// TIA Portal project "Project2" (V20)

(* hardware
DEVICE "S71500/ET200MP station_1"  S7-1500 station
   slot 0: "Rail_0"  Rack  6ES7 590-1***0-0AA0
   slot 1: "PLC_1"  CPU 1511-1 PN  6ES7 511-1AK00-0AB0  V1.8
      slot 3: "CPU display_1"  6ES7591-1AA00-0AA0
DEVICE "PC-System_1"  SIMATIC PC station
   slot 0: "SIMATIC PC station"  Rail  SIMATIC PC-Station  V1.0
      slot 125: "Stationmanager"  Station_Manager  V6.0.4
   slot 1: "HMI_RT_1"  WinCC RT Advanced  6AV2 104-0xxxx-xxxx  17.0.0.0
      slot 33792: "Computer interface"  Host interface
   slot 2: "IE general_1"  IE General  IE_CP  V8.2.0
      slot 1: "PROFINET interface"  IEGeneral.Interface.8.2.0
*)

// ===== PLC "PLC_1"  CPU 1511-1 PN =====

VAR_GLOBAL   // PLC tag table "Default tag table"
   "Brake_En" AT %M0.0 : Bool;
   "Baffle_Out" AT %MW18 : Int;
   "RPM_In" AT %MW2 : Int;
   "OilTemp_In" AT %MW4 : Int;
   "Baffle_En" AT %M0.1 : Bool;
   "Current_In" AT %MW6 : Int;
   "OilPumpVFDsp_Out" AT %MW8 : Int;
   "OilPumpVFDen_Out" AT %M0.2 : Bool;
   "OilFlow_In" AT %MW10 : Int;
   "TriggerSCL" AT %M0.4 : Bool;
   "Program_Lang" AT %MW12 : Int;
   "Button_LAD" AT %M0.3 : Bool;
   "Button_FBD" AT %M0.5 : Bool;
   "Button_SCL" AT %M0.6 : Bool;
   "Button_STL" AT %M0.7 : Bool;
   "TriggerLAD" AT %M1.0 : Bool;
   "TriggerFBD" AT %M1.1 : Bool;
   "TriggerSTL" AT %M1.2 : Bool;
   "AlarmHorn_En" AT %M1.3 : Bool;
   "StationInterlock_En" AT %M1.4 : Bool;
   "Baffle_Percent" AT %MW14 : Int;
   "OilPumpVFD_percent" AT %MW16 : Int;
   "RPM" AT %MW20 : Int;
   "OilFlow" AT %MW24 : Int;
   "OilTemp" AT %MW28 : Int;
   "Current" AT %MW22 : Int;
   "Static_Test" AT %M1.5 : Bool;
   "BaffleOff_Button" AT %M1.6 : Bool;
   "BaffleHand_Button" AT %M1.7 : Bool;
   "BaffleAuto_Button" AT %M26.0 : Bool;
   "Baffle_HOA" AT %MW70 : Int;
   "SiOff_Button" AT %M26.1 : Bool;
   "StationInterlock_HOA" AT %MW30 : Int;
   "SiHand_Button" AT %M26.2 : Bool;
   "SiAuto_Button" AT %M26.3 : Bool;
   "Brake_HOA" AT %MW40 : Int;
   "BrakeOff_Button" AT %M26.4 : Bool;
   "BrakeHand_Button" AT %M26.5 : Bool;
   "BrakeAuto_Button" AT %M26.6 : Bool;
   "AlarmHorn_HOA" AT %MW50 : Int;
   "AlarmHornOff_Button" AT %M26.7 : Bool;
   "AlarmHornHand_Button" AT %M34.0 : Bool;
   "AlarmHornAuto_Button" AT %M34.1 : Bool;
   "OilPump_HOA" AT %MW60 : Int;
   "OilPumpOff_Button" AT %M34.2 : Bool;
   "OilPumpHand_Button" AT %M34.3 : Bool;
   "OilPumpAuto_Button" AT %M34.4 : Bool;
   "Baffle_Ctrl" AT %M34.5 : Bool;
   "OilPump_Ctrl" AT %M37.0 : Bool;
   "AlarmHorn_Ctrl" AT %M37.1 : Bool;
   "Brake_Ctrl" AT %M37.2 : Bool;
   "StationInterlock_Ctrl" AT %M37.3 : Bool;
   "SeqRunning" AT %M90.0 : Bool;
   "SeqStart" AT %M90.1 : Bool;
   "trigger1" AT %M90.2 : Bool;
   "trigger2" AT %M90.3 : Bool;
   "OverrideVFD_Set" AT %MW92 : Int;
END_VAR

VAR_GLOBAL   // PLC tag table "Alarm_Tags"
   "Overcurrent_set" AT %MW32 : Int;
   "Alarm_Reset" AT %M27.0 : Bool;
   "Alarm_Mute" AT %M27.1 : Bool;
   "OverCurrent_DelaySec" AT %MW38 : Int;
   "OverCurrent_Alarm" AT %M27.2 : Bool;
   "OverCurrent_Horn" AT %M27.3 : Bool;
   "HiOilTemp_DelaySec" AT %MW42 : Int;
   "OilTempMax_set" AT %MW44 : Int;
   "OilTempMax_Horn" AT %M27.4 : Bool;
   "OilTempMax_Alarm" AT %M27.5 : Bool;
   "OverSpeed_DelaySec" AT %MW46 : Int;
   "Overspeed_set" AT %MW48 : Int;
   "OverSpeed_Horn" AT %M27.7 : Bool;
   "OverSpeed_Alarm" AT %M34.6 : Bool;
   "MinOil_set" AT %MW54 : Int;
   "LowOil_Horn" AT %M34.7 : Bool;
   "LowOil_Alarm" AT %M35.0 : Bool;
   "LowOil_DelaySec" AT %MW52 : Int;
   "HighOil_DelaySec" AT %MW56 : Int;
   "MaxOil_set" AT %MW58 : Int;
   "HighOil_Horn" AT %M35.1 : Bool;
   "HighOil_Alarm" AT %M35.2 : Bool;
   "EStop" AT %M35.3 : Bool;
   "EStop_Horn" AT %M35.4 : Bool;
   "EStop_Alarm" AT %M35.5 : Bool;
   "BrakeFail_DelaySec" AT %MW62 : Int;
   "BrakeFail_Horn" AT %M35.6 : Bool;
   "BrakeFail_Alarm" AT %M35.7 : Bool;
END_VAR

VAR_GLOBAL   // PLC tag table "Modes_Tags"
   "WarmupMode" AT %M27.6 : Bool;
   "IdleMode" AT %M36.3 : Bool;
   "GenerationMode" AT %M36.1 : Bool;
   "StabilizeMode" AT %M36.0 : Bool;
   "CooldownMode" AT %M36.2 : Bool;
   "FaultMode" AT %M36.4 : Bool;
   "WarmupRPM" AT %MW64 : Int;
   "Baffel_PID_Set" AT %MW66 : Int;
   "WarmupPumpPct" AT %MW68 : Int;
   "Oilpump_Set" AT %MW72 : Int;
   "WarmupOilTemp" AT %MW74 : Int;
   "WarmupOilTemp_DelaySet" AT %MW76 : Int;
   "WarmupTrans" AT %M36.5 : Bool;
   "Baffel_PID_In" AT %MW78 : Int;
   "Stabile_Current_Set" AT %MW80 : Int;
   "Stabilize_Current_Delay_Set" AT %MW82 : Int;
   "StabilizeTrans" AT %M36.6 : Bool;
   "SystemStop_Button" AT %M36.7 : Bool;
   "GenerationTrans" AT %M37.4 : Bool;
   "SystemStart_Button" AT %M37.5 : Bool;
   "Start_Seq" AT %M37.6 : Bool;
   "CooldownTrans" AT %M37.7 : Bool;
   "CoolDownOilTemp_DelaySet" AT %MW84 : Int;
   "CoolDownRPM_Set" AT %MW86 : Int;
   "CoolDownOilTemp" AT %MW88 : Int;
END_VAR

DATA_BLOCK "SimLogic_DB"   // DB1
{ S7_Optimized_Access := 'TRUE' }
VERSION : 0.1
// stored: InstanceOfName SimLogic
"SimLogic"
BEGIN
END_DATA_BLOCK

DATA_BLOCK "LAD_HOA_DB"   // DB2
{ S7_Optimized_Access := 'TRUE' }
VERSION : 0.1
// stored: InstanceOfName LAD_HOA
"LAD_HOA"
BEGIN
END_DATA_BLOCK

DATA_BLOCK "LAD_IO_DB"   // DB4
{ S7_Optimized_Access := 'TRUE' }
VERSION : 0.1
// stored: InstanceOfName LAD_IO
"LAD_IO"
BEGIN
END_DATA_BLOCK

DATA_BLOCK "FBD_IO_DB"   // DB5
{ S7_Optimized_Access := 'TRUE' }
VERSION : 0.1
// stored: InstanceOfName FBD_IO
"FBD_IO"
BEGIN
END_DATA_BLOCK

DATA_BLOCK "SCL_IO_DB"   // DB6
{ S7_Optimized_Access := 'TRUE' }
VERSION : 0.1
// stored: InstanceOfName SCL_IO
"SCL_IO"
BEGIN
END_DATA_BLOCK

DATA_BLOCK "STL_IO_DB"   // DB7
{ S7_Optimized_Access := 'TRUE' }
VERSION : 0.1
// stored: InstanceOfName STL_IO
"STL_IO"
BEGIN
END_DATA_BLOCK

DATA_BLOCK "FBD_HOA_DB"   // DB8
{ S7_Optimized_Access := 'TRUE' }
VERSION : 0.1
// stored: InstanceOfName FBD_HOA
"FBD_HOA"
BEGIN
END_DATA_BLOCK

DATA_BLOCK "SCL_HOA_DB"   // DB9
{ S7_Optimized_Access := 'TRUE' }
VERSION : 0.1
// stored: InstanceOfName SCL_HOA
"SCL_HOA"
BEGIN
END_DATA_BLOCK

DATA_BLOCK "STL_HOA_DB"   // DB10
{ S7_Optimized_Access := 'TRUE' }
VERSION : 0.1
// stored: InstanceOfName STL_HOA
"STL_HOA"
BEGIN
END_DATA_BLOCK

DATA_BLOCK "LAD_Alarm_DB"   // DB11
{ S7_Optimized_Access := 'TRUE' }
VERSION : 0.1
// stored: InstanceOfName LAD_Alarm
"LAD_Alarm"
BEGIN
END_DATA_BLOCK

DATA_BLOCK "FBD_Alarm_DB"   // DB20
{ S7_Optimized_Access := 'TRUE' }
VERSION : 0.1
// stored: InstanceOfName FBD_Alarm
"FBD_Alarm"
BEGIN
END_DATA_BLOCK

DATA_BLOCK "SCL_Alarm_DB"   // DB21
{ S7_Optimized_Access := 'TRUE' }
VERSION : 0.1
// stored: InstanceOfName SCL_Alarm
"SCL_Alarm"
BEGIN
END_DATA_BLOCK

DATA_BLOCK "STL_Alarm_DB"   // DB22
{ S7_Optimized_Access := 'TRUE' }
VERSION : 0.1
// stored: InstanceOfName STL_Alarm
"STL_Alarm"
BEGIN
END_DATA_BLOCK

DATA_BLOCK "LAD_Modes_DB"   // DB25
{ S7_Optimized_Access := 'TRUE' }
VERSION : 0.1
// stored: InstanceOfName LAD_Modes
"LAD_Modes"
BEGIN
END_DATA_BLOCK

DATA_BLOCK "SEQ_DB"   // DB26
{ S7_Optimized_Access := 'TRUE' }
VERSION : 0.1
// stored: InstanceOfName SEQ
"SEQ"
BEGIN
END_DATA_BLOCK

// folder: System blocks/Program resources

DATA_BLOCK "IEC_Timer_0_DB_25"   // DB3
{ S7_Optimized_Access := 'TRUE' }
AUTHOR : Simatic
FAMILY : IEC
NAME : IEC_TMR
VERSION : 1.0
// stored: InstanceOfName IEC_TIMER
"IEC_TIMER"
BEGIN
END_DATA_BLOCK

DATA_BLOCK "OverCurrent_Tolerance"   // DB12
{ S7_Optimized_Access := 'TRUE' }
AUTHOR : Simatic
FAMILY : IEC
NAME : IEC_TMR
VERSION : 1.0
// stored: InstanceOfName IEC_TIMER
"IEC_TIMER"
BEGIN
END_DATA_BLOCK

DATA_BLOCK "OilTempHi_Tolerance"   // DB13
{ S7_Optimized_Access := 'TRUE' }
AUTHOR : Simatic
FAMILY : IEC
NAME : IEC_TMR
VERSION : 1.0
// stored: InstanceOfName IEC_TIMER
"IEC_TIMER"
BEGIN
END_DATA_BLOCK

DATA_BLOCK "OverSpeed_Tolerance"   // DB14
{ S7_Optimized_Access := 'TRUE' }
AUTHOR : Simatic
FAMILY : IEC
NAME : IEC_TMR
VERSION : 1.0
// stored: InstanceOfName IEC_TIMER
"IEC_TIMER"
BEGIN
END_DATA_BLOCK

DATA_BLOCK "OilLow_Tolerance"   // DB15
{ S7_Optimized_Access := 'TRUE' }
AUTHOR : Simatic
FAMILY : IEC
NAME : IEC_TMR
VERSION : 1.0
// stored: InstanceOfName IEC_TIMER
"IEC_TIMER"
BEGIN
END_DATA_BLOCK

DATA_BLOCK "OilHigh_Tolerance"   // DB16
{ S7_Optimized_Access := 'TRUE' }
AUTHOR : Simatic
FAMILY : IEC
NAME : IEC_TMR
VERSION : 1.0
// stored: InstanceOfName IEC_TIMER
"IEC_TIMER"
BEGIN
END_DATA_BLOCK

DATA_BLOCK "IEC_Timer_0_DB"   // DB17
{ S7_Optimized_Access := 'TRUE' }
AUTHOR : Simatic
FAMILY : IEC
NAME : IEC_TMR
VERSION : 1.0
// stored: InstanceOfName IEC_TIMER
"IEC_TIMER"
BEGIN
END_DATA_BLOCK

DATA_BLOCK "Warmup_to_Stable"   // DB18
{ S7_Optimized_Access := 'TRUE' }
AUTHOR : Simatic
FAMILY : IEC
NAME : IEC_TMR
VERSION : 1.0
// stored: InstanceOfName IEC_TIMER
"IEC_TIMER"
BEGIN
END_DATA_BLOCK

DATA_BLOCK "BrakeFail_Tolerance"   // DB19
{ S7_Optimized_Access := 'TRUE' }
AUTHOR : Simatic
FAMILY : IEC
NAME : IEC_TMR
VERSION : 1.0
// stored: InstanceOfName IEC_TIMER
"IEC_TIMER"
BEGIN
END_DATA_BLOCK

DATA_BLOCK "Stabilize_To_Generation"   // DB23
{ S7_Optimized_Access := 'TRUE' }
AUTHOR : Simatic
FAMILY : IEC
NAME : IEC_TMR
VERSION : 1.0
// stored: InstanceOfName IEC_TIMER
"IEC_TIMER"
BEGIN
END_DATA_BLOCK

DATA_BLOCK "Stable_To_Idle"   // DB24
{ S7_Optimized_Access := 'TRUE' }
AUTHOR : Simatic
FAMILY : IEC
NAME : IEC_TMR
VERSION : 1.0
// stored: InstanceOfName IEC_TIMER
"IEC_TIMER"
BEGIN
END_DATA_BLOCK

DATA_BLOCK "IEC_Timer_1_DB"   // DB43
{ S7_Optimized_Access := 'TRUE' }
AUTHOR : Simatic
FAMILY : IEC
NAME : IEC_TMR
VERSION : 1.0
// stored: InstanceOfName IEC_TIMER
"IEC_TIMER"
BEGIN
END_DATA_BLOCK

// folder: (top level)

FUNCTION_BLOCK "SimLogic"   // FB1, FBD
{ S7_Optimized_Access := 'TRUE' }
VERSION : 0.1
   VAR
      "TO" : Bool;
      rpmv : Int;
      addrpmv : Bool;
      otsp : Int;
      ott : Int;
      TO1 : Bool;
      TO2 : Bool;
      be2 : Int;
      be3 : Int;
      be1 : Int;
      TO3 : Bool;
   END_VAR
   VAR_TEMP
      bf : Int;
      rpmvt : Int;
      bfr : Real;
   END_VAR
BEGIN

REGION Network 1
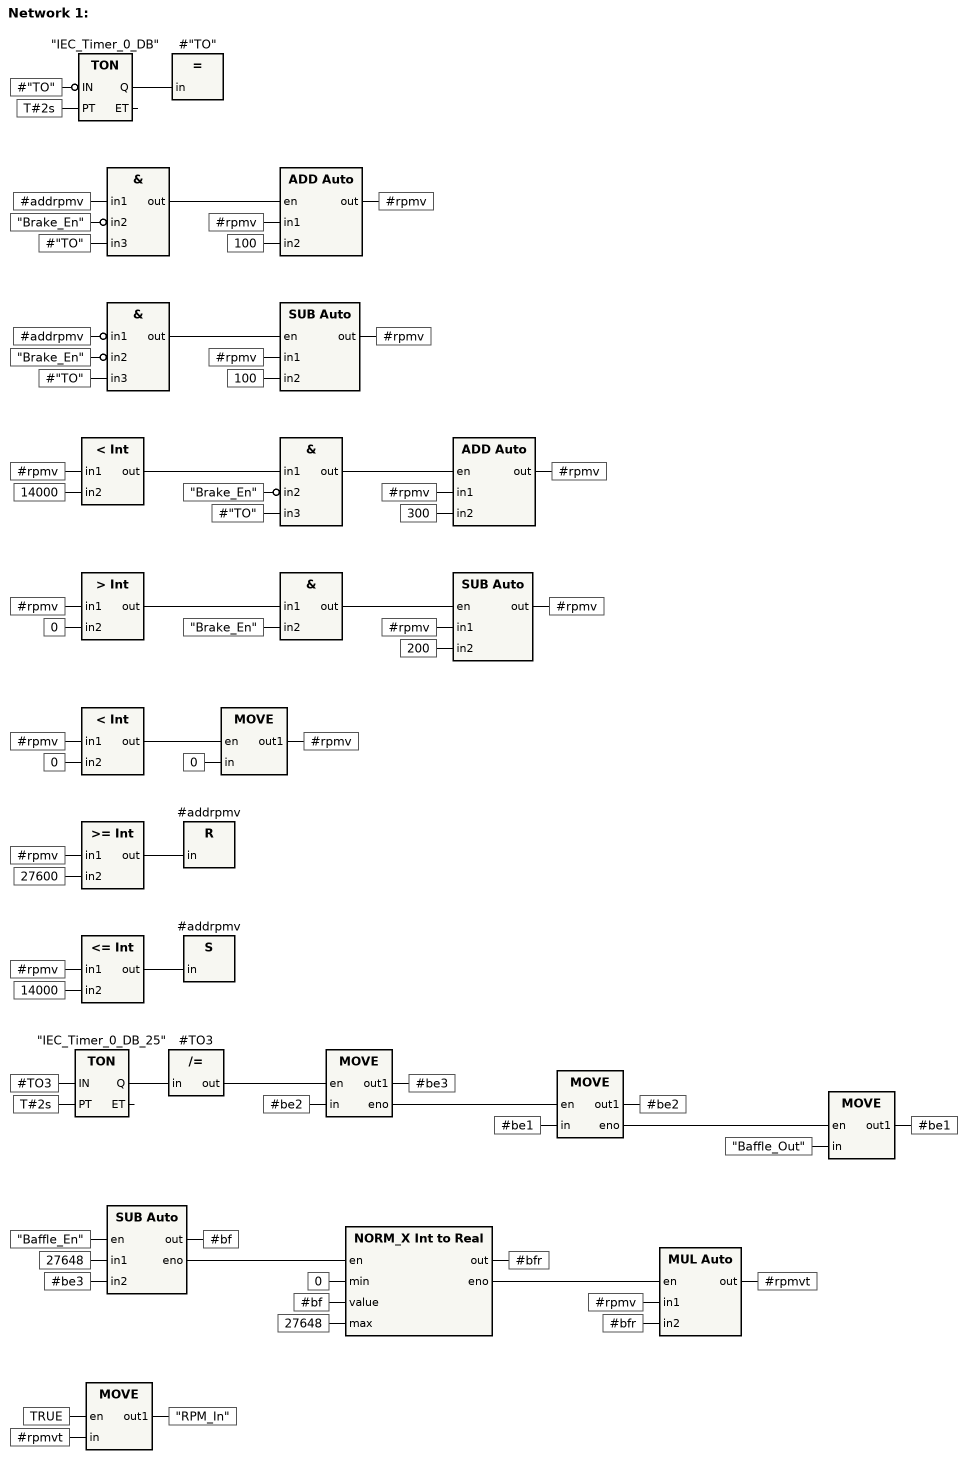
   "IEC_Timer_0_DB".TON(IN := NOT #"TO", PT := T#2s);
   #"TO" := "IEC_Timer_0_DB".Q;
   IF #addrpmv AND NOT "Brake_En" AND #"TO" THEN #rpmv := #rpmv + 100; END_IF;
   IF NOT #addrpmv AND NOT "Brake_En" AND #"TO" THEN #rpmv := #rpmv - 100; END_IF;
   IF (#rpmv < 14000) AND NOT "Brake_En" AND #"TO" THEN #rpmv := #rpmv + 300; END_IF;
   IF (#rpmv > 0) AND "Brake_En" THEN #rpmv := #rpmv - 200; END_IF;
   IF #rpmv < 0 THEN #rpmv := 0; END_IF;
   IF #rpmv >= 27600 THEN #addrpmv := FALSE; END_IF;
   IF #rpmv <= 14000 THEN #addrpmv := TRUE; END_IF;
   "IEC_Timer_0_DB_25".TON(IN := #TO3, PT := T#2s);
   #TO3 := NOT "IEC_Timer_0_DB_25".Q;
   IF "IEC_Timer_0_DB_25".Q THEN
       #be3 := #be2;
       #be2 := #be1;
       #be1 := "Baffle_Out";
   END_IF;
   IF "Baffle_En" THEN
       #bf := 27648 - #be3;
       #bfr := NORM_X(MIN := 0, VALUE := #bf, MAX := 27648);
       #rpmvt := #rpmv * #bfr;
   END_IF;
   IF TRUE THEN "RPM_In" := #rpmvt; END_IF;
END_REGION

REGION Network 2
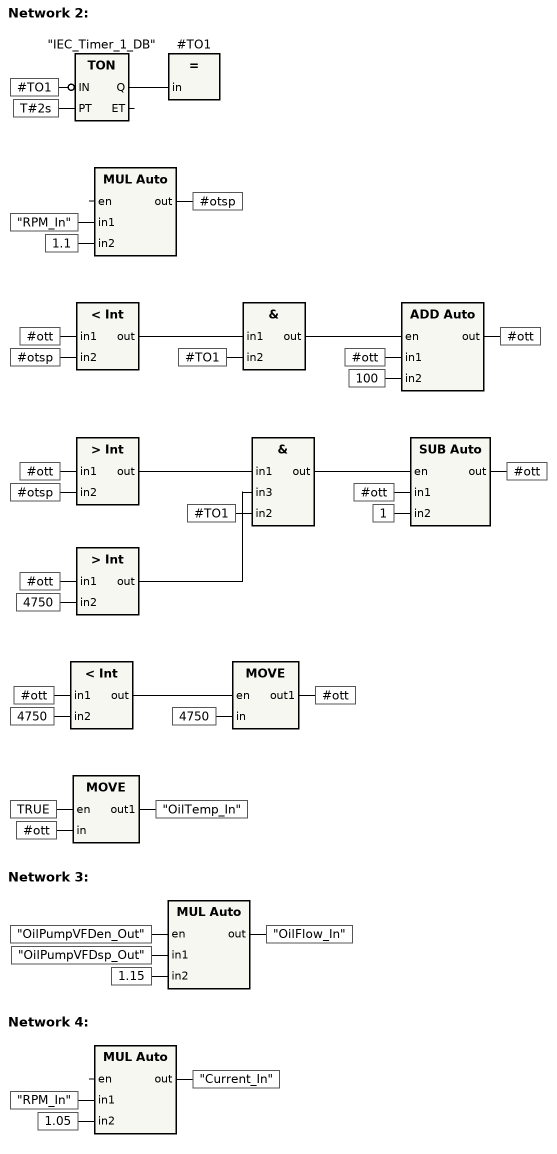
   "IEC_Timer_1_DB".TON(IN := NOT #TO1, PT := T#2s);
   #TO1 := "IEC_Timer_1_DB".Q;
   #otsp := "RPM_In" * 1.1;
   IF (#ott < #otsp) AND #TO1 THEN #ott := #ott + 100; END_IF;
   IF (#ott > #otsp) AND (#ott > 4750) AND #TO1 THEN #ott := #ott - 1; END_IF;
   IF #ott < 4750 THEN #ott := 4750; END_IF;
   IF TRUE THEN "OilTemp_In" := #ott; END_IF;
END_REGION

REGION Network 3
   IF "OilPumpVFDen_Out" THEN "OilFlow_In" := "OilPumpVFDsp_Out" * 1.15; END_IF;
END_REGION

REGION Network 4
   "Current_In" := "RPM_In" * 1.05;
END_REGION
END_FUNCTION_BLOCK

FUNCTION_BLOCK "LAD_IO"   // FB2, LAD
TITLE = I/O logic of the controller in Ladder Diagram
{ S7_Optimized_Access := 'TRUE' }
VERSION : 0.1
// Here are the outputs/output logic of the controller programmed.
BEGIN

REGION Network 1: Digital Outputs
   // Enable logic of DQs, enables when either hand-mode or auto-mode is chosen.
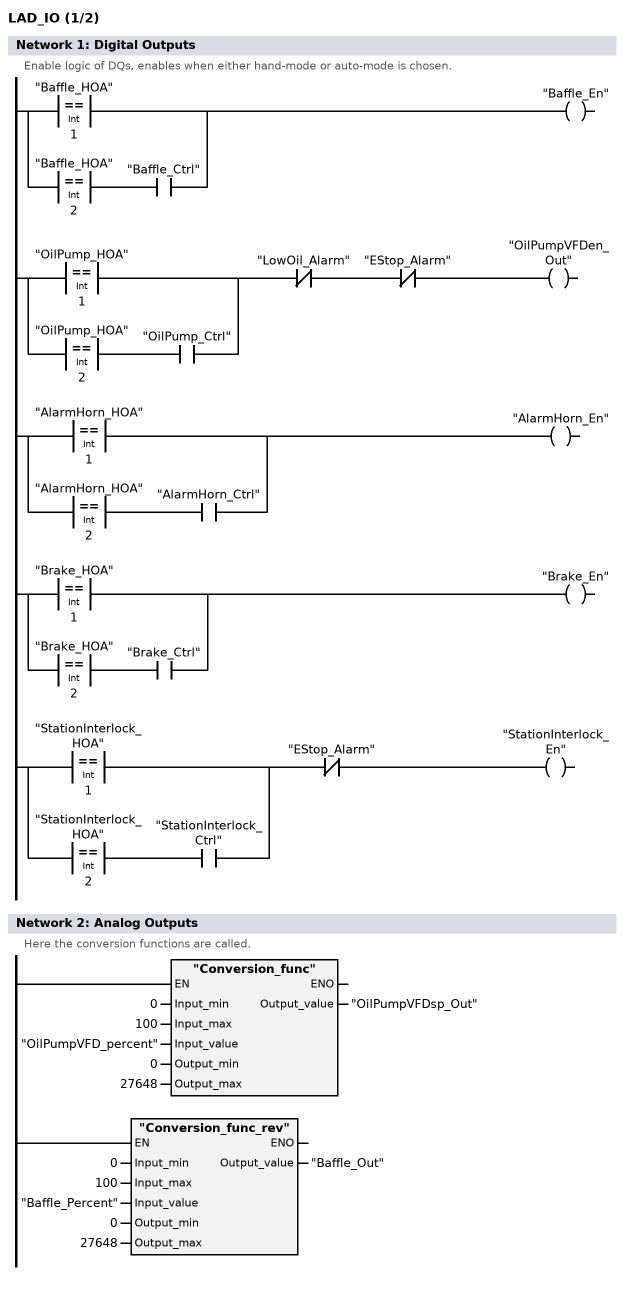
   RUNG wire#powerrail
      { S7_Templates := "SrcType := Int" } EQ_Contact(in1 := "Baffle_HOA", in2 := 1)
      wire#w1
      Coil( "Baffle_En" )
   END_RUNG
   RUNG wire#powerrail
      { S7_Templates := "SrcType := Int" } EQ_Contact(in1 := "Baffle_HOA", in2 := 2)
      Contact( "Baffle_Ctrl" )
   END_RUNG wire#w1
   RUNG wire#powerrail
      { S7_Templates := "SrcType := Int" } EQ_Contact(in1 := "OilPump_HOA", in2 := 1)
      wire#w2
      I_Contact( "LowOil_Alarm" )
      I_Contact( "EStop_Alarm" )
      Coil( "OilPumpVFDen_Out" )
   END_RUNG
   RUNG wire#powerrail
      { S7_Templates := "SrcType := Int" } EQ_Contact(in1 := "OilPump_HOA", in2 := 2)
      Contact( "OilPump_Ctrl" )
   END_RUNG wire#w2
   RUNG wire#powerrail
      { S7_Templates := "SrcType := Int" } EQ_Contact(in1 := "AlarmHorn_HOA", in2 := 1)
      wire#w3
      Coil( "AlarmHorn_En" )
   END_RUNG
   RUNG wire#powerrail
      { S7_Templates := "SrcType := Int" } EQ_Contact(in1 := "AlarmHorn_HOA", in2 := 2)
      Contact( "AlarmHorn_Ctrl" )
   END_RUNG wire#w3
   RUNG wire#powerrail
      { S7_Templates := "SrcType := Int" } EQ_Contact(in1 := "Brake_HOA", in2 := 1)
      wire#w4
      Coil( "Brake_En" )
   END_RUNG
   RUNG wire#powerrail
      { S7_Templates := "SrcType := Int" } EQ_Contact(in1 := "Brake_HOA", in2 := 2)
      Contact( "Brake_Ctrl" )
   END_RUNG wire#w4
   RUNG wire#powerrail
      { S7_Templates := "SrcType := Int" } EQ_Contact(in1 := "StationInterlock_HOA", in2 := 1)
      wire#w5
      I_Contact( "EStop_Alarm" )
      Coil( "StationInterlock_En" )
   END_RUNG
   RUNG wire#powerrail
      { S7_Templates := "SrcType := Int" } EQ_Contact(in1 := "StationInterlock_HOA", in2 := 2)
      Contact( "StationInterlock_Ctrl" )
   END_RUNG wire#w5
   // the same network as SCL:
   "Baffle_En" := ("Baffle_HOA" = 1) OR (("Baffle_HOA" = 2) AND "Baffle_Ctrl");
   "OilPumpVFDen_Out" := (("OilPump_HOA" = 1) OR (("OilPump_HOA" = 2) AND "OilPump_Ctrl")) AND NOT "LowOil_Alarm" AND NOT "EStop_Alarm";
   "AlarmHorn_En" := ("AlarmHorn_HOA" = 1) OR (("AlarmHorn_HOA" = 2) AND "AlarmHorn_Ctrl");
   "Brake_En" := ("Brake_HOA" = 1) OR (("Brake_HOA" = 2) AND "Brake_Ctrl");
   "StationInterlock_En" := (("StationInterlock_HOA" = 1) OR (("StationInterlock_HOA" = 2) AND "StationInterlock_Ctrl")) AND NOT "EStop_Alarm";
END_REGION

REGION Network 2: Analog Outputs
   // Here the conversion functions are called.
   RUNG wire#powerrail
      "Conversion_func"(Input_min := 0, Input_max := 100, Input_value := "OilPumpVFD_percent", Output_min := 0, Output_max := 27648, Output_value => "OilPumpVFDsp_Out")
   END_RUNG
   RUNG wire#powerrail
      "Conversion_func_rev"(Input_min := 0, Input_max := 100, Input_value := "Baffle_Percent", Output_min := 0, Output_max := 27648, Output_value => "Baffle_Out")
   END_RUNG
   // the same network as SCL:
   "Conversion_func"(Input_min := 0,
                     Input_max := 100,
                     Input_value := "OilPumpVFD_percent",
                     Output_min := 0,
                     Output_max := 27648,
                     Output_value => "OilPumpVFDsp_Out");
   "Conversion_func_rev"(Input_min := 0,
                         Input_max := 100,
                         Input_value := "Baffle_Percent",
                         Output_min := 0,
                         Output_max := 27648,
                         Output_value => "Baffle_Out");
END_REGION

REGION Network 3: Analog Inputs
   // Here the conversion functions are called as well.
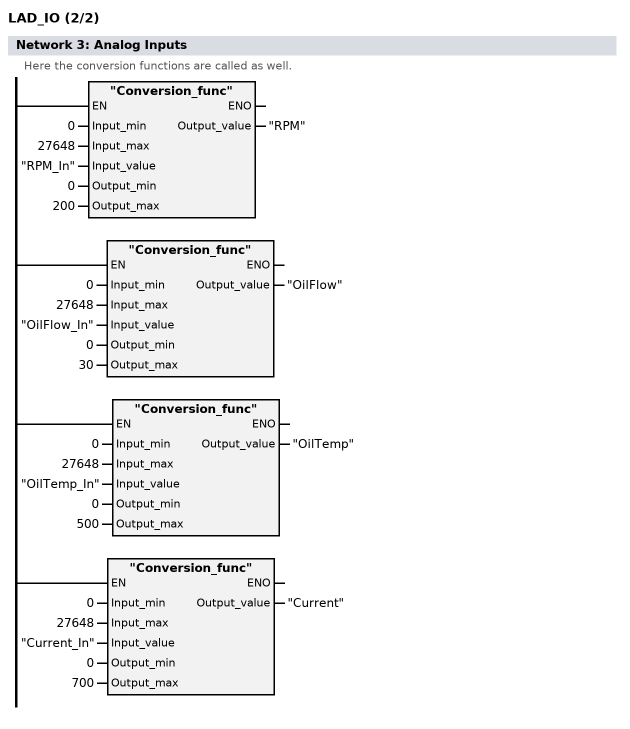
   RUNG wire#powerrail
      "Conversion_func"(Input_min := 0, Input_max := 27648, Input_value := "RPM_In", Output_min := 0, Output_max := 200, Output_value => "RPM")
   END_RUNG
   RUNG wire#powerrail
      "Conversion_func"(Input_min := 0, Input_max := 27648, Input_value := "OilFlow_In", Output_min := 0, Output_max := 30, Output_value => "OilFlow")
   END_RUNG
   RUNG wire#powerrail
      "Conversion_func"(Input_min := 0, Input_max := 27648, Input_value := "OilTemp_In", Output_min := 0, Output_max := 500, Output_value => "OilTemp")
   END_RUNG
   RUNG wire#powerrail
      "Conversion_func"(Input_min := 0, Input_max := 27648, Input_value := "Current_In", Output_min := 0, Output_max := 700, Output_value => "Current")
   END_RUNG
   // the same network as SCL:
   "Conversion_func"(Input_min := 0,
                     Input_max := 27648,
                     Input_value := "RPM_In",
                     Output_min := 0,
                     Output_max := 200,
                     Output_value => "RPM");
   "Conversion_func"(Input_min := 0,
                     Input_max := 27648,
                     Input_value := "OilFlow_In",
                     Output_min := 0,
                     Output_max := 30,
                     Output_value => "OilFlow");
   "Conversion_func"(Input_min := 0,
                     Input_max := 27648,
                     Input_value := "OilTemp_In",
                     Output_min := 0,
                     Output_max := 500,
                     Output_value => "OilTemp");
   "Conversion_func"(Input_min := 0,
                     Input_max := 27648,
                     Input_value := "Current_In",
                     Output_min := 0,
                     Output_max := 700,
                     Output_value => "Current");
END_REGION
END_FUNCTION_BLOCK

FUNCTION_BLOCK "FBD_IO"   // FB3, FBD
TITLE = I/O logic of the controller in Function Block Diagram
{ S7_Optimized_Access := 'TRUE' }
VERSION : 0.1
// Here are the outputs/output logic of the controller programmed.
BEGIN

REGION Network 1: Digital Outputs
   // Enable logic of DQs
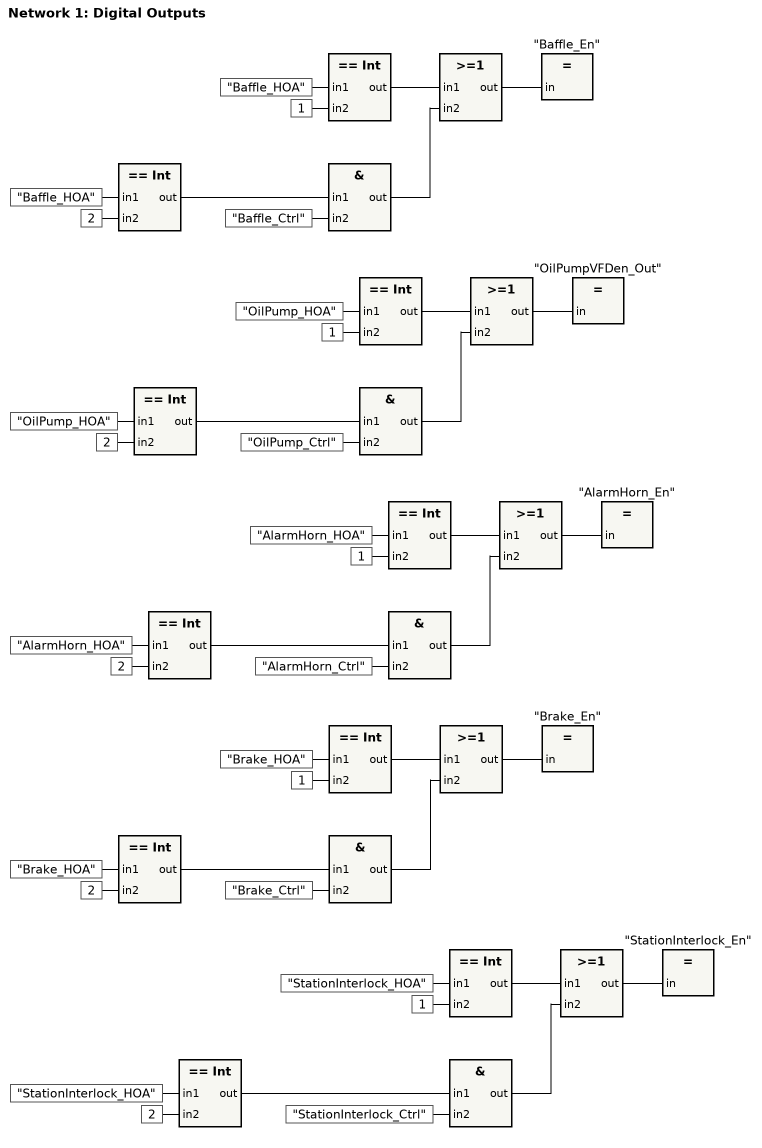
   "Baffle_En" := ("Baffle_HOA" = 1) OR (("Baffle_HOA" = 2) AND "Baffle_Ctrl");
   "OilPumpVFDen_Out" := ("OilPump_HOA" = 1) OR (("OilPump_HOA" = 2) AND "OilPump_Ctrl");
   "AlarmHorn_En" := ("AlarmHorn_HOA" = 1) OR (("AlarmHorn_HOA" = 2) AND "AlarmHorn_Ctrl");
   "Brake_En" := ("Brake_HOA" = 1) OR (("Brake_HOA" = 2) AND "Brake_Ctrl");
   "StationInterlock_En" := ("StationInterlock_HOA" = 1) OR (("StationInterlock_HOA" = 2) AND "StationInterlock_Ctrl");
END_REGION

REGION Network 2: Analog Outputs
   // Here the conversion functions are called.
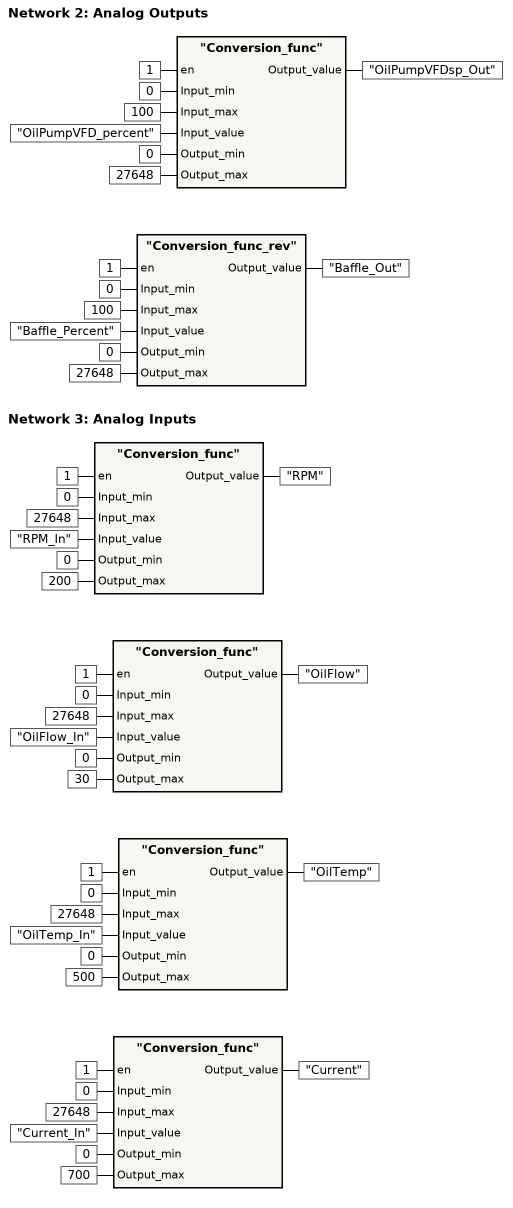
   IF 1 THEN
       "Conversion_func"(Input_min := 0,
                         Input_max := 100,
                         Input_value := "OilPumpVFD_percent",
                         Output_min := 0,
                         Output_max := 27648,
                         Output_value => "OilPumpVFDsp_Out");
       "Conversion_func_rev"(Input_min := 0,
                             Input_max := 100,
                             Input_value := "Baffle_Percent",
                             Output_min := 0,
                             Output_max := 27648,
                             Output_value => "Baffle_Out");
   END_IF;
END_REGION

REGION Network 3: Analog Inputs
   // Here the conversion functions are called as well.
   IF 1 THEN
       "Conversion_func"(Input_min := 0,
                         Input_max := 27648,
                         Input_value := "RPM_In",
                         Output_min := 0,
                         Output_max := 200,
                         Output_value => "RPM");
       "Conversion_func"(Input_min := 0,
                         Input_max := 27648,
                         Input_value := "OilFlow_In",
                         Output_min := 0,
                         Output_max := 30,
                         Output_value => "OilFlow");
       "Conversion_func"(Input_min := 0,
                         Input_max := 27648,
                         Input_value := "OilTemp_In",
                         Output_min := 0,
                         Output_max := 500,
                         Output_value => "OilTemp");
       "Conversion_func"(Input_min := 0,
                         Input_max := 27648,
                         Input_value := "Current_In",
                         Output_min := 0,
                         Output_max := 700,
                         Output_value => "Current");
   END_IF;
END_REGION
END_FUNCTION_BLOCK

FUNCTION_BLOCK "SCL_IO"   // FB4, SCL
{ S7_Optimized_Access := 'TRUE' }
VERSION : 0.1
BEGIN
   (*
   I/O logic OF the controller in Structured Control Languege: Here are the outputs/output logic OF the controller programmed.
   *)

   (*Digital Outputs: Enable logic OF DQs*)
   IF "Baffle_HOA" = 0 OR ("Baffle_HOA" = 2 AND NOT "Baffle_Ctrl") THEN
       // disable
       "Baffle_En" := 0;
   END_IF;
   IF "Baffle_HOA" = 1 OR ("Baffle_HOA" = 2 AND "Baffle_Ctrl") THEN
       // enable
       "Baffle_En" := 1;
   END_IF;

   IF "OilPump_HOA" = 0 OR ("OilPump_HOA" = 2 AND NOT "OilPump_Ctrl") THEN
       "OilPumpVFDen_Out" := 0;
   END_IF;
   IF "OilPump_HOA" = 1 OR ("OilPump_HOA" = 2 AND "OilPump_Ctrl") THEN
       "OilPumpVFDen_Out" := 1;
   END_IF;

   IF "AlarmHorn_HOA" = 0 OR ("AlarmHorn_HOA" = 2 AND NOT "AlarmHorn_Ctrl") THEN
       "AlarmHorn_En" := 0;
   END_IF;
   IF "AlarmHorn_HOA" = 1 OR ("AlarmHorn_HOA" = 2 AND "AlarmHorn_Ctrl") THEN
       "AlarmHorn_En" := 1;
   END_IF;

   IF "Brake_HOA" = 0 OR ("Brake_HOA" = 2 AND NOT "Brake_Ctrl") THEN
       "Brake_En" := 0;
   END_IF;
   IF "Brake_HOA" = 1 OR ("Brake_HOA" = 2 AND "Brake_Ctrl") THEN
       "Brake_En" := 1;
   END_IF;

   IF "StationInterlock_HOA" = 0 OR ("StationInterlock_HOA" = 2 AND NOT "StationInterlock_Ctrl") THEN
       "StationInterlock_En" := 0;
   END_IF;
   IF "StationInterlock_HOA" = 1 OR ("StationInterlock_HOA" = 2 AND "StationInterlock_Ctrl") THEN
       "StationInterlock_En" := 1;
   END_IF;

   (*Analog Outputs: conversion functions are called*)
   "Conversion_func"(Input_min:=0,
                     Input_max:=100,
                     Input_value:="OilPumpVFD_percent",
                     Output_min:=0,
                     Output_max:=27648,
                     Output_value=>"OilPumpVFDsp_Out");
   "Conversion_func_rev"(Input_min:=0,
                         Input_max:=100,
                         Input_value:="Baffle_Percent",
                         Output_min:=0,
                         Output_max:=27648,
                         Output_value=>"Baffle_Out");

   (*Analog Inputs: conversion functions are called as well*)
   "Conversion_func"(Input_min:=0,
                     Input_max:=27648,
                     Input_value:="RPM_In",
                     Output_min:=0,
                     Output_max:=200,
                     Output_value=>"RPM");
   "Conversion_func"(Input_min := 0,
                     Input_max := 27648,
                     Input_value := "OilFlow_In",
                     Output_min := 0,
                     Output_max := 30,
                     Output_value => "OilFlow");
   "Conversion_func"(Input_min := 0,
                     Input_max := 27648,
                     Input_value := "OilTemp_In",
                     Output_min := 0,
                     Output_max := 500,
                     Output_value => "OilTemp");
   "Conversion_func"(Input_min := 0,
                     Input_max := 27648,
                     Input_value := "Current_In",
                     Output_min := 0,
                     Output_max := 700,
                     Output_value => "Current");
END_FUNCTION_BLOCK

FUNCTION_BLOCK "STL_IO"   // FB5, STL
TITLE = I/O logic of the controller in STL
{ S7_Optimized_Access := 'TRUE' }
VERSION : 0.1
// Here are the outputs/output logic of the controller programmed.
BEGIN

REGION Network 1: Digital Outputs
   // Enable logic of DQs
   //Baffle
         L     "Baffle_HOA";
         L     1;
         ==I;
         O(;
         L     "Baffle_HOA";
         L     2;
         ==I;
         A     "Baffle_Ctrl";
         );
         =     "Baffle_En";

   //OilPump
         L     "OilPump_HOA";
         L     0;
         ==I;
         O(;
         L     "OilPump_HOA";
         L     2;
         ==I;
         AN    "OilPump_Ctrl";
         );
         R     "OilPumpVFDen_Out";

         L     "OilPump_HOA";
         L     1;
         ==I;
         O(;
         L     "OilPump_HOA";
         L     2;
         ==I;
         A     "OilPump_Ctrl";
         );
         S     "OilPumpVFDen_Out";

   //AlarmHorn
         L     "AlarmHorn_HOA";
         L     0;
         ==I;
         O(;
         L     "AlarmHorn_HOA";
         L     2;
         ==I;
         AN    "AlarmHorn_Ctrl";
         );
         R     "AlarmHorn_En";

         L     "AlarmHorn_HOA";
         L     1;
         ==I;
         O(;
         L     "AlarmHorn_HOA";
         L     2;
         ==I;
         A     "AlarmHorn_Ctrl";
         );
         S     "AlarmHorn_En";

   //Brake
         L     "Brake_HOA";
         L     0;
         ==I;
         O(;
         L     "Brake_HOA";
         L     2;
         ==I;
         AN    "Brake_Ctrl";
         );
         R     "Brake_En";

         L     "Brake_HOA";
         L     1;
         ==I;
         O(;
         L     "Brake_HOA";
         L     2;
         ==I;
         A     "Brake_Ctrl";
         );
         S     "Brake_En";

   //StationInterlock
         L     "StationInterlock_HOA";
         L     0;
         ==I;
         O(;
         L     "StationInterlock_HOA";
         L     2;
         ==I;
         AN    "StationInterlock_Ctrl";
         );
         R     "StationInterlock_En";

         L     "StationInterlock_HOA";
         L     1;
         ==I;
         O(;
         L     "StationInterlock_HOA";
         L     2;
         ==I;
         A     "StationInterlock_Ctrl";
         );
         S     "StationInterlock_En";
END_REGION

REGION Network 2: Analog Outputs
   // Here the conversion functions are called.
         CALL  "Conversion_func"
         ( Input_min    := 0,
           Input_max    := 100,
           Input_value  := "OilPumpVFD_percent",
           Output_min   := 0,
           Output_max   := 27648,
           Output_value := "OilPumpVFDsp_Out"
         );

         CALL  "Conversion_func_rev"
         ( Input_min    := 0,
           Input_max    := 100,
           Input_value  := "Baffle_Percent",
           Output_min   := 0,
           Output_max   := 27648,
           Output_value := "Baffle_Out"
         );
END_REGION

REGION Network 3: Analog Inputs
   // Here the conversion functions are called as well.
         CALL  "Conversion_func"
         ( Input_min    := 0,
           Input_max    := 27648,
           Input_value  := "RPM_In",
           Output_min   := 0,
           Output_max   := 200,
           Output_value := "RPM"
         );

         CALL  "Conversion_func"
         ( Input_min    := 0,
           Input_max    := 27648,
           Input_value  := "OilFlow_In",
           Output_min   := 0,
           Output_max   := 30,
           Output_value := "OilFlow"
         );

         CALL  "Conversion_func"
         ( Input_min    := 0,
           Input_max    := 27648,
           Input_value  := "OilTemp_In",
           Output_min   := 0,
           Output_max   := 500,
           Output_value := "OilTemp"
         );

         CALL  "Conversion_func"
         ( Input_min    := 0,
           Input_max    := 27648,
           Input_value  := "Current_In",
           Output_min   := 0,
           Output_max   := 700,
           Output_value := "Current"
         );
END_REGION
END_FUNCTION_BLOCK

FUNCTION_BLOCK "LAD_HOA"   // FB6, LAD
TITLE = HOA value setting in ladder diagram
{ S7_Optimized_Access := 'TRUE' }
VERSION : 0.1
// HOA only for the digital outputs. Analog outputs automatically controlled by PID.
   VAR
      TG1 : Bool;
      TG2 : Bool;
      TG3 : Bool;
      TG4 : Bool;
      TG5 : Bool;
      TG6 : Bool;
      TG7 : Bool;
      TG8 : Bool;
      TG9 : Bool;
      TG10 : Bool;
      TG11 : Bool;
      TG12 : Bool;
      TG13 : Bool;
      TG14 : Bool;
      TG15 : Bool;
   END_VAR
   VAR_TEMP   // added for the SCL form of the ladder/FBD networks
      _w1 : Bool;
      _w2 : Bool;
      _w3 : Bool;
   END_VAR
BEGIN

REGION Network 1: Baffle HOA
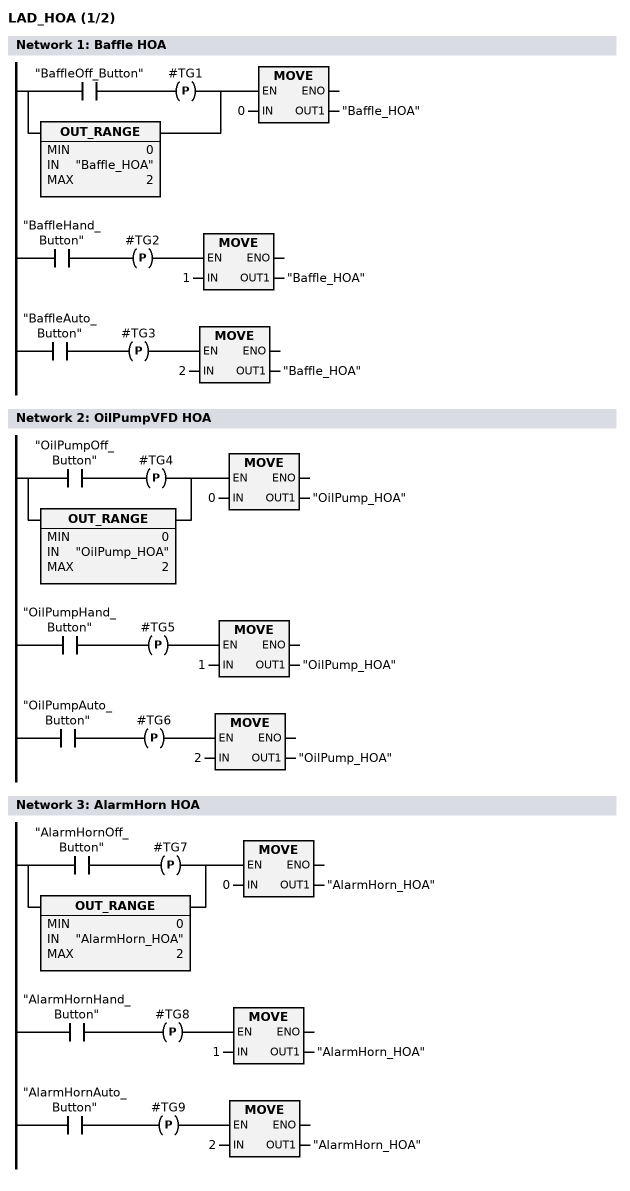
   #_w1 := "BaffleOff_Button" AND NOT #TG1;   // rising edge
   #TG1 := "BaffleOff_Button";
   IF #_w1 OR ("Baffle_HOA" < 0) OR ("Baffle_HOA" > 2) THEN "Baffle_HOA" := 0; END_IF;
   #_w2 := "BaffleHand_Button" AND NOT #TG2;   // rising edge
   #TG2 := "BaffleHand_Button";
   IF #_w2 THEN "Baffle_HOA" := 1; END_IF;
   #_w3 := "BaffleAuto_Button" AND NOT #TG3;   // rising edge
   #TG3 := "BaffleAuto_Button";
   IF #_w3 THEN "Baffle_HOA" := 2; END_IF;
END_REGION

REGION Network 2: OilPumpVFD HOA
   #_w1 := "OilPumpOff_Button" AND NOT #TG4;   // rising edge
   #TG4 := "OilPumpOff_Button";
   IF #_w1 OR ("OilPump_HOA" < 0) OR ("OilPump_HOA" > 2) THEN "OilPump_HOA" := 0; END_IF;
   #_w2 := "OilPumpHand_Button" AND NOT #TG5;   // rising edge
   #TG5 := "OilPumpHand_Button";
   IF #_w2 THEN "OilPump_HOA" := 1; END_IF;
   #_w3 := "OilPumpAuto_Button" AND NOT #TG6;   // rising edge
   #TG6 := "OilPumpAuto_Button";
   IF #_w3 THEN "OilPump_HOA" := 2; END_IF;
END_REGION

REGION Network 3: AlarmHorn HOA
   #_w1 := "AlarmHornOff_Button" AND NOT #TG7;   // rising edge
   #TG7 := "AlarmHornOff_Button";
   IF #_w1 OR ("AlarmHorn_HOA" < 0) OR ("AlarmHorn_HOA" > 2) THEN "AlarmHorn_HOA" := 0; END_IF;
   #_w2 := "AlarmHornHand_Button" AND NOT #TG8;   // rising edge
   #TG8 := "AlarmHornHand_Button";
   IF #_w2 THEN "AlarmHorn_HOA" := 1; END_IF;
   #_w3 := "AlarmHornAuto_Button" AND NOT #TG9;   // rising edge
   #TG9 := "AlarmHornAuto_Button";
   IF #_w3 THEN "AlarmHorn_HOA" := 2; END_IF;
END_REGION

REGION Network 4: Brake HOA
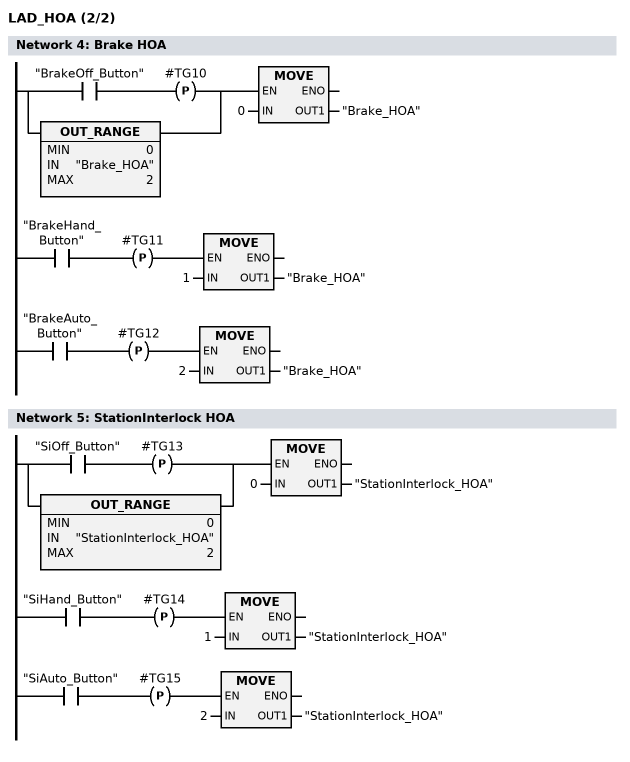
   #_w1 := "BrakeOff_Button" AND NOT #TG10;   // rising edge
   #TG10 := "BrakeOff_Button";
   IF #_w1 OR ("Brake_HOA" < 0) OR ("Brake_HOA" > 2) THEN "Brake_HOA" := 0; END_IF;
   #_w2 := "BrakeHand_Button" AND NOT #TG11;   // rising edge
   #TG11 := "BrakeHand_Button";
   IF #_w2 THEN "Brake_HOA" := 1; END_IF;
   #_w3 := "BrakeAuto_Button" AND NOT #TG12;   // rising edge
   #TG12 := "BrakeAuto_Button";
   IF #_w3 THEN "Brake_HOA" := 2; END_IF;
END_REGION

REGION Network 5: StationInterlock HOA
   #_w1 := "SiOff_Button" AND NOT #TG13;   // rising edge
   #TG13 := "SiOff_Button";
   IF #_w1 OR ("StationInterlock_HOA" < 0) OR ("StationInterlock_HOA" > 2) THEN
       "StationInterlock_HOA" := 0;
   END_IF;
   #_w2 := "SiHand_Button" AND NOT #TG14;   // rising edge
   #TG14 := "SiHand_Button";
   IF #_w2 THEN "StationInterlock_HOA" := 1; END_IF;
   #_w3 := "SiAuto_Button" AND NOT #TG15;   // rising edge
   #TG15 := "SiAuto_Button";
   IF #_w3 THEN "StationInterlock_HOA" := 2; END_IF;
END_REGION
END_FUNCTION_BLOCK

FUNCTION_BLOCK "FBD_HOA"   // FB7, FBD
TITLE = HOA value setting in Function Block diagram
{ S7_Optimized_Access := 'TRUE' }
VERSION : 0.1
// HOA only for the digital outputs. Analog outputs automatically controlled by PID.
   VAR
      TG_0 : Bool;
      TG_1 : Bool;
      TG_2 : Bool;
      TG_3 : Bool;
      TG_4 : Bool;
      TG_5 : Bool;
      TG_6 : Bool;
      TG_7 : Bool;
      TG_8 : Bool;
      TG_9 : Bool;
      TG_10 : Bool;
      TG_11 : Bool;
      TG_12 : Bool;
      TG_13 : Bool;
      TG_14 : Bool;
   END_VAR
   VAR_TEMP   // added for the SCL form of the ladder/FBD networks
      _w1 : Bool;
      _w2 : Bool;
      _w3 : Bool;
   END_VAR
BEGIN

REGION Network 1: Baffle HOA
   // Baffel_HOA
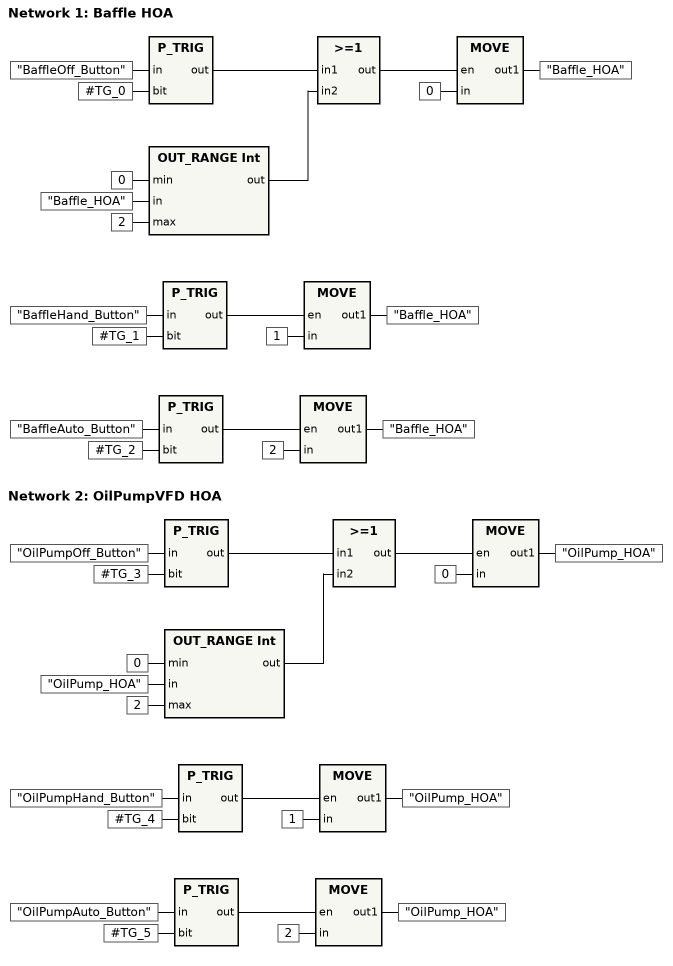
   #_w1 := "BaffleOff_Button" AND NOT #TG_0;   // rising edge
   #TG_0 := "BaffleOff_Button";
   IF #_w1 OR ("Baffle_HOA" < 0) OR ("Baffle_HOA" > 2) THEN "Baffle_HOA" := 0; END_IF;
   #_w2 := "BaffleHand_Button" AND NOT #TG_1;   // rising edge
   #TG_1 := "BaffleHand_Button";
   IF #_w2 THEN "Baffle_HOA" := 1; END_IF;
   #_w3 := "BaffleAuto_Button" AND NOT #TG_2;   // rising edge
   #TG_2 := "BaffleAuto_Button";
   IF #_w3 THEN "Baffle_HOA" := 2; END_IF;
END_REGION

REGION Network 2: OilPumpVFD HOA
   #_w1 := "OilPumpOff_Button" AND NOT #TG_3;   // rising edge
   #TG_3 := "OilPumpOff_Button";
   IF #_w1 OR ("OilPump_HOA" < 0) OR ("OilPump_HOA" > 2) THEN "OilPump_HOA" := 0; END_IF;
   #_w2 := "OilPumpHand_Button" AND NOT #TG_4;   // rising edge
   #TG_4 := "OilPumpHand_Button";
   IF #_w2 THEN "OilPump_HOA" := 1; END_IF;
   #_w3 := "OilPumpAuto_Button" AND NOT #TG_5;   // rising edge
   #TG_5 := "OilPumpAuto_Button";
   IF #_w3 THEN "OilPump_HOA" := 2; END_IF;
END_REGION

REGION Network 3: AlarmHorn HOA
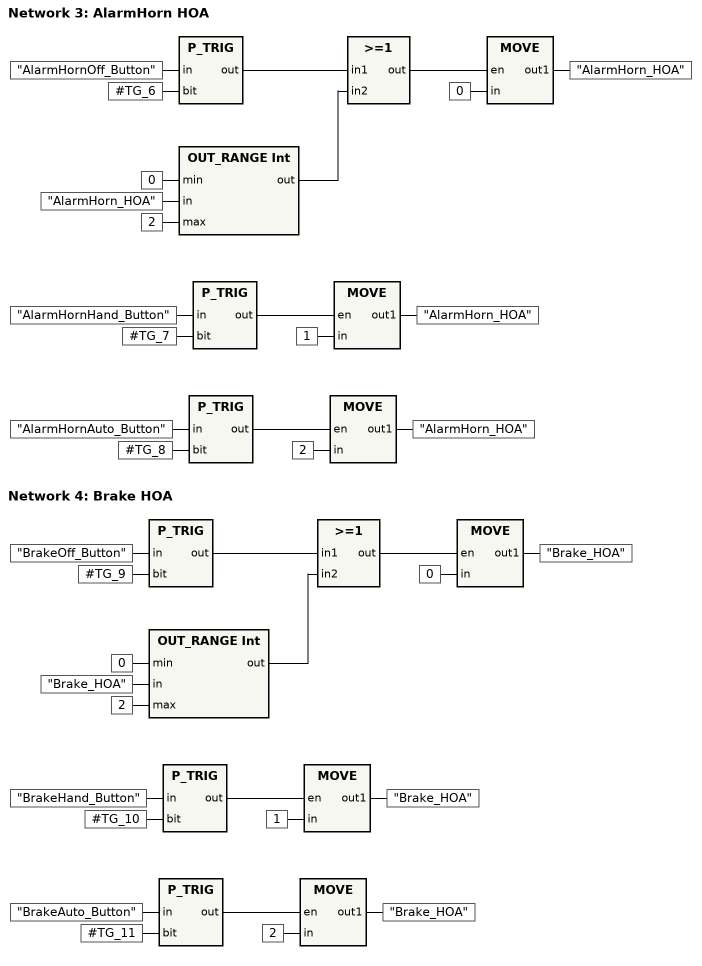
   #_w1 := "AlarmHornOff_Button" AND NOT #TG_6;   // rising edge
   #TG_6 := "AlarmHornOff_Button";
   IF #_w1 OR ("AlarmHorn_HOA" < 0) OR ("AlarmHorn_HOA" > 2) THEN "AlarmHorn_HOA" := 0; END_IF;
   #_w2 := "AlarmHornHand_Button" AND NOT #TG_7;   // rising edge
   #TG_7 := "AlarmHornHand_Button";
   IF #_w2 THEN "AlarmHorn_HOA" := 1; END_IF;
   #_w3 := "AlarmHornAuto_Button" AND NOT #TG_8;   // rising edge
   #TG_8 := "AlarmHornAuto_Button";
   IF #_w3 THEN "AlarmHorn_HOA" := 2; END_IF;
END_REGION

REGION Network 4: Brake HOA
   #_w1 := "BrakeOff_Button" AND NOT #TG_9;   // rising edge
   #TG_9 := "BrakeOff_Button";
   IF #_w1 OR ("Brake_HOA" < 0) OR ("Brake_HOA" > 2) THEN "Brake_HOA" := 0; END_IF;
   #_w2 := "BrakeHand_Button" AND NOT #TG_10;   // rising edge
   #TG_10 := "BrakeHand_Button";
   IF #_w2 THEN "Brake_HOA" := 1; END_IF;
   #_w3 := "BrakeAuto_Button" AND NOT #TG_11;   // rising edge
   #TG_11 := "BrakeAuto_Button";
   IF #_w3 THEN "Brake_HOA" := 2; END_IF;
END_REGION

REGION Network 5: StationInterlock HOA
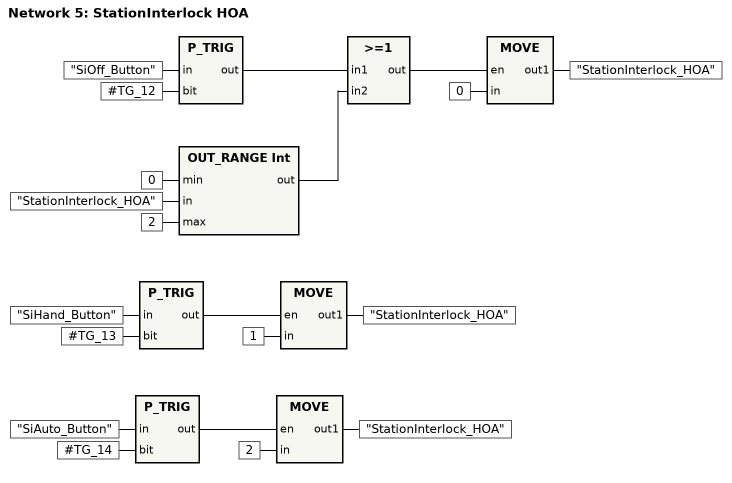
   #_w1 := "SiOff_Button" AND NOT #TG_12;   // rising edge
   #TG_12 := "SiOff_Button";
   IF #_w1 OR ("StationInterlock_HOA" < 0) OR ("StationInterlock_HOA" > 2) THEN
       "StationInterlock_HOA" := 0;
   END_IF;
   #_w2 := "SiHand_Button" AND NOT #TG_13;   // rising edge
   #TG_13 := "SiHand_Button";
   IF #_w2 THEN "StationInterlock_HOA" := 1; END_IF;
   #_w3 := "SiAuto_Button" AND NOT #TG_14;   // rising edge
   #TG_14 := "SiAuto_Button";
   IF #_w3 THEN "StationInterlock_HOA" := 2; END_IF;
END_REGION
END_FUNCTION_BLOCK

FUNCTION_BLOCK "SCL_HOA"   // FB8, SCL
{ S7_Optimized_Access := 'TRUE' }
VERSION : 0.1
   VAR
      BaffleOffTrig : R_TRIG;
      BaffleHandTrig : R_TRIG;
      BaffleAutoTrig : R_TRIG;
      PumpOffTrig : R_TRIG;
      PumpHandTrig : R_TRIG;
      PumpAutoTrig : R_TRIG;
      AlarmOffTrig : R_TRIG;
      AlarmHandTrig : R_TRIG;
      AlarmAutoTrig : R_TRIG;
      BrakeOffTrig : R_TRIG;
      BrakeHandTrig : R_TRIG;
      BrakeAutoTrig : R_TRIG;
      SiOffTrig : R_TRIG;
      SiHandTrig : R_TRIG;
      SiAutoTrig : R_TRIG;
   END_VAR
BEGIN
   // HOA value setting in Structured control language

   //Baffle HOA
   #BaffleOffTrig(CLK := "BaffleOff_Button");
   #BaffleHandTrig(CLK := "BaffleHand_Button");
   #BaffleAutoTrig(CLK := "BaffleAuto_Button");

   IF "Baffle_HOA" >2 OR "Baffle_HOA" <0 THEN
       // FaultMode, HOA Off
       "Baffle_HOA" := 0;
   END_IF;

   IF #BaffleOffTrig.Q THEN
       // OffMode
       "Baffle_HOA" := 0;
   ELSIF #BaffleHandTrig.Q THEN
       // HandMode
       "Baffle_HOA" := 1;
   ELSIF #BaffleAutoTrig.Q THEN
       // AutoMode
       "Baffle_HOA" := 2;
   END_IF;


   //OilPumpVFD HOA
   #PumpOffTrig(CLK := "OilPumpOff_Button");
   #PumpHandTrig(CLK := "OilPumpHand_Button");
   #PumpAutoTrig(CLK := "OilPumpAuto_Button");

   IF "OilPump_HOA" > 2 OR "OilPump_HOA" < 0 THEN
       // FaultMode, HOA Off
       "OilPump_HOA" := 0;
   END_IF;

   IF #PumpOffTrig.Q THEN
       // OffMode
       "OilPump_HOA" := 0;
   ELSIF #PumpHandTrig.Q THEN
       // HandMode
       "OilPump_HOA" := 1;
   ELSIF #PumpAutoTrig.Q THEN
       // AutoMode
       "OilPump_HOA" := 2;
   END_IF;


   //AlarmHorn HOA
   #AlarmOffTrig(CLK := "AlarmHornOff_Button");
   #AlarmHandTrig(CLK := "AlarmHornHand_Button");
   #AlarmAutoTrig(CLK := "AlarmHornAuto_Button");

   IF "AlarmHorn_HOA" > 2 OR "AlarmHorn_HOA" < 0 THEN
       // FaultMode, HOA Off
       "AlarmHorn_HOA" := 0;
   END_IF;

   IF #AlarmOffTrig.Q THEN
       // OffMode
       "AlarmHorn_HOA" := 0;
   ELSIF #AlarmHandTrig.Q THEN
       // HandMode
       "AlarmHorn_HOA" := 1;
   ELSIF #AlarmAutoTrig.Q THEN
       // AutoMode
       "AlarmHorn_HOA" := 2;
   END_IF;


   //Brake HOA
   #BrakeOffTrig(CLK := "BrakeOff_Button");
   #BrakeHandTrig(CLK := "BrakeHand_Button");
   #BrakeAutoTrig(CLK := "BrakeAuto_Button");

   IF "Brake_HOA" > 2 OR "Brake_HOA" < 0 THEN
       // FaultMode, HOA Off
       "Brake_HOA" := 0;
   END_IF;

   IF #BrakeOffTrig.Q THEN
       // OffMode
       "Brake_HOA" := 0;
   ELSIF #BrakeHandTrig.Q THEN
       // HandMode
       "Brake_HOA" := 1;
   ELSIF #BrakeAutoTrig.Q THEN
       // AutoMode
       "Brake_HOA" := 2;
   END_IF;


   //StationInterlock HOA
   #SiOffTrig(CLK := "SiOff_Button");
   #SiHandTrig(CLK := "SiHand_Button");
   #SiAutoTrig(CLK := "SiAuto_Button");

   IF "StationInterlock_HOA" > 2 OR "StationInterlock_HOA" < 0 THEN
       // FaultMode, HOA Off
       "StationInterlock_HOA" := 0;
   END_IF;

   IF #SiOffTrig.Q THEN
       // OffMode
       "StationInterlock_HOA" := 0;
   ELSIF #SiHandTrig.Q THEN
       // HandMode
       "StationInterlock_HOA" := 1;
   ELSIF #SiAutoTrig.Q THEN
       // AutoMode
       "StationInterlock_HOA" := 2;
   END_IF;
END_FUNCTION_BLOCK

FUNCTION_BLOCK "STL_HOA"   // FB9, STL
TITLE = HOA value setting in STL
{ S7_Optimized_Access := 'TRUE' }
VERSION : 0.1
   VAR
      BaffleOffTrig : Bool;
      BaffleHandTrig : Bool;
      BaffleAutoTrig : Bool;
      PumpOffTrig : Bool;
      PumpHandTrig : Bool;
      PumpAutoTrig : Bool;
      AlarmOffTrig : Bool;
      AlarmHandTrig : Bool;
      AlarmAutoTrig : Bool;
      BrakeOffTrig : Bool;
      BrakeHandTrig : Bool;
      BrakeAutoTrig : Bool;
      SiOffTrig : Bool;
      SiHandTrig : Bool;
      SiAutoTrig : Bool;
   END_VAR
BEGIN

REGION Network 1: Baffel HOA
         L     "Baffle_HOA";
         L     0;
         <I;
         JC    Baffel_HOA_Off;
         CLR;

         L     "Baffle_HOA";
         L     2;
         >I;
         JC    Baffel_HOA_Off;
         CLR;

         A     "BaffleOff_Button";
         FP    #BaffleOffTrig;
         JC    Baffel_HOA_Off;

         A     "BaffleHand_Button";
         FP    #BaffleHandTrig;
         JC    Baffel_HOA_Hand;

         A     "BaffleAuto_Button";
         FP    #BaffleAutoTrig;
         JC    Baffel_HOA_Auto;

   // Idle. In a scan period no buttons are newly pressed, then jump to next network.
         JU    OilPump;

   Baffel_HOA_Off:L     0;
         T     "Baffle_HOA";
         JU    OilPump;
   Baffel_HOA_Hand:L     1;
         T     "Baffle_HOA";
         JU    OilPump;
   Baffel_HOA_Auto:L     2;
         T     "Baffle_HOA";
         JU    OilPump;
END_REGION

REGION Network 2: Oilpump HOA
   OilPump:L     "OilPump_HOA";
         L     0;
         <I;
         JC    OilPump_HOA_Off;
         CLR;

         L     "OilPump_HOA";
         L     2;
         >I;
         JC    OilPump_HOA_Off;
         CLR;

         A     "OilPumpOff_Button";
         FP    #PumpOffTrig;
         JC    OilPump_HOA_Off;

         A     "OilPumpHand_Button";
         FP    #PumpHandTrig;
         JC    OilPump_HOA_Hand;

         A     "OilPumpAuto_Button";
         FP    #PumpAutoTrig;
         JC    OilPump_HOA_Auto;

         JU    AlarmHorn;

   OilPump_HOA_Off:L     0;
         T     "OilPump_HOA";
         JU    AlarmHorn;
   OilPump_HOA_Hand:L     1;
         T     "OilPump_HOA";
         JU    AlarmHorn;
   OilPump_HOA_Auto:L     2;
         T     "OilPump_HOA";
         JU    AlarmHorn;
END_REGION

REGION Network 3: AlarmHorn HOA
   AlarmHorn:L     "AlarmHorn_HOA";
         L     0;
         <I;
         JC    AlarmHorn_HOA_Off;
         CLR;

         L     "AlarmHorn_HOA";
         L     2;
         >I;
         JC    AlarmHorn_HOA_Off;
         CLR;

         A     "AlarmHornOff_Button";
         FP    #AlarmOffTrig;
         JC    AlarmHorn_HOA_Off;

         A     "AlarmHornHand_Button";
         FP    #AlarmHandTrig;
         JC    AlarmHorn_HOA_Hand;

         A     "AlarmHornAuto_Button";
         FP    #AlarmAutoTrig;
         JC    AlarmHorn_HOA_Auto;

         JU    Brake;

   AlarmHorn_HOA_Off:L     0;
         T     "AlarmHorn_HOA";
         JU    Brake;
   AlarmHorn_HOA_Hand:L     1;
         T     "AlarmHorn_HOA";
         JU    Brake;
   AlarmHorn_HOA_Auto:L     2;
         T     "AlarmHorn_HOA";
         JU    Brake;
END_REGION

REGION Network 4: Brake HOA
   Brake:L     "Brake_HOA";
         L     0;
         <I;
         JC    Brake_HOA_Off;
         CLR;

         L     "Brake_HOA";
         L     2;
         >I;
         JC    Brake_HOA_Off;
         CLR;

         A     "BrakeOff_Button";
         FP    #BrakeOffTrig;
         JC    Brake_HOA_Off;

         A     "BrakeHand_Button";
         FP    #BrakeHandTrig;
         JC    Brake_HOA_Hand;

         A     "BrakeAuto_Button";
         FP    #BrakeAutoTrig;
         JC    Brake_HOA_Auto;

         JU    StationInterlock;

   Brake_HOA_Off:L     0;
         T     "Brake_HOA";
         JU    StationInterlock;
   Brake_HOA_Hand:L     1;
         T     "Brake_HOA";
         JU    StationInterlock;
   Brake_HOA_Auto:L     2;
         T     "Brake_HOA";
         JU    StationInterlock;
END_REGION

REGION Network 5: StationInterlock HOA
   StationInterlock:L     "StationInterlock_HOA";
         L     0;
         <I;
         JC    StationInterlock_HOA_Off;
         CLR;

         L     "StationInterlock_HOA";
         L     2;
         >I;
         JC    StationInterlock_HOA_Off;
         CLR;

         A     "SiOff_Button";
         FP    #SiOffTrig;
         JC    StationInterlock_HOA_Off;

         A     "SiHand_Button";
         FP    #SiHandTrig;
         JC    StationInterlock_HOA_Hand;

         A     "SiAuto_Button";
         FP    #SiAutoTrig;
         JC    StationInterlock_HOA_Auto;

         JU    End;

   StationInterlock_HOA_Off:L     0;
         T     "StationInterlock_HOA";
         JU    End;
   StationInterlock_HOA_Hand:L     1;
         T     "StationInterlock_HOA";
         JU    End;
   StationInterlock_HOA_Auto:L     2;
         T     "StationInterlock_HOA";
         JU    End;

   End:  BE;
END_REGION
END_FUNCTION_BLOCK

FUNCTION_BLOCK "LAD_Alarm"   // FB10, LAD
TITLE = Alarms in LAD
{ S7_Optimized_Access := 'TRUE' }
VERSION : 0.1
// When any alarm is triggered, the alert horn will sound. 
// The tolerance time of each alarm can be modified individually. 
// MUL is used to convert sec to ms. MOVE is used to force datatype convert.
   VAR
      Trigger1 : Bool;
      Trigger2 : Bool;
      Trigger3 : Bool;
      Trigger4 : Bool;
      Trigger5 : Bool;
      Trigger6 : Bool;
      Trigger7 : Bool;
   END_VAR
   VAR_TEMP
      OC_delay : Int;
      tv1 : Time;
      OverCurrent_Trigger : Bool;
      HT_delay : Int;
      tv2 : Time;
      OilTempMax_Trigger : Bool;
      OS_delay : Int;
      tv3 : Time;
      OverSpeed_Trigger : Bool;
      OL_delay : Int;
      tv4 : Time;
      LowOil_Trigger : Bool;
      OH_delay : Int;
      tv5 : Time;
      HighOil_Trigger : Bool;
      EStop_Trigger : Bool;
      BF_delay : Int;
      tv6 : Time;
      BF_Trigger : Bool;
   END_VAR
   VAR_TEMP   // added for the SCL form of the ladder/FBD networks
      _w1 : Bool;
      _w2 : Bool;
   END_VAR
BEGIN

REGION Network 1: Overcurrent Alarm
   // Activate when current exceeds the Max setpoint.
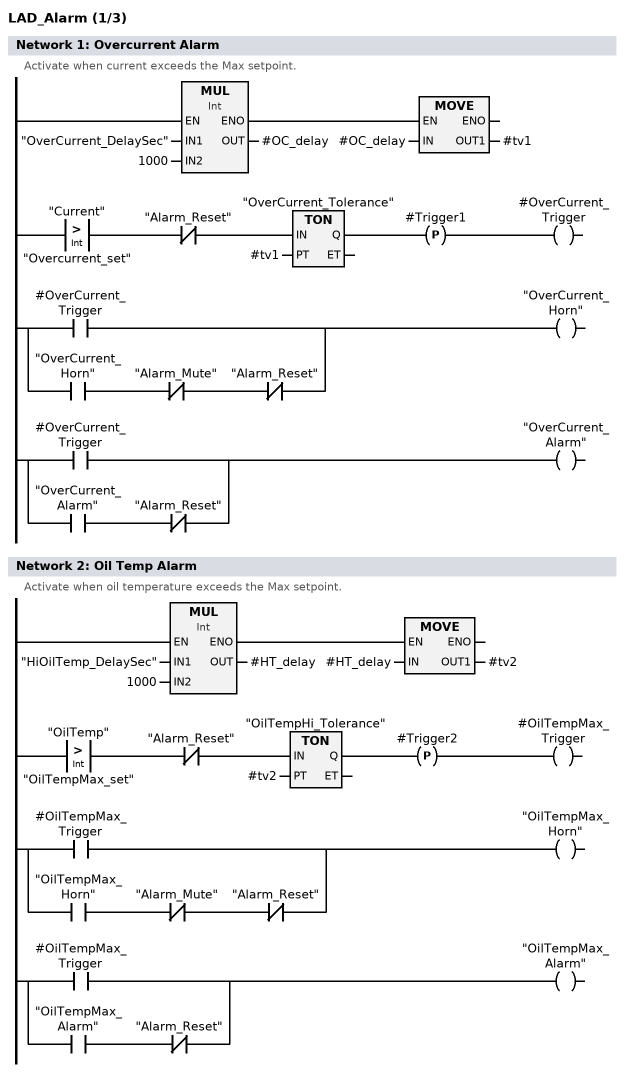
   #OC_delay := "OverCurrent_DelaySec" * 1000;
   #tv1 := #OC_delay;
   "OverCurrent_Tolerance".TON(IN := ("Current" > "Overcurrent_set") AND NOT "Alarm_Reset", PT := #tv1);
   #_w1 := "OverCurrent_Tolerance".Q AND NOT #Trigger1;   // rising edge
   #Trigger1 := "OverCurrent_Tolerance".Q;
   #OverCurrent_Trigger := #_w1;
   "OverCurrent_Horn" := #OverCurrent_Trigger OR ("OverCurrent_Horn" AND NOT "Alarm_Mute" AND NOT "Alarm_Reset");
   "OverCurrent_Alarm" := #OverCurrent_Trigger OR ("OverCurrent_Alarm" AND NOT "Alarm_Reset");
END_REGION

REGION Network 2: Oil Temp Alarm
   // Activate when oil temperature exceeds the Max setpoint.
   #HT_delay := "HiOilTemp_DelaySec" * 1000;
   #tv2 := #HT_delay;
   "OilTempHi_Tolerance".TON(IN := ("OilTemp" > "OilTempMax_set") AND NOT "Alarm_Reset", PT := #tv2);
   #_w1 := "OilTempHi_Tolerance".Q AND NOT #Trigger2;   // rising edge
   #Trigger2 := "OilTempHi_Tolerance".Q;
   #OilTempMax_Trigger := #_w1;
   "OilTempMax_Horn" := #OilTempMax_Trigger OR ("OilTempMax_Horn" AND NOT "Alarm_Mute" AND NOT "Alarm_Reset");
   "OilTempMax_Alarm" := #OilTempMax_Trigger OR ("OilTempMax_Alarm" AND NOT "Alarm_Reset");
END_REGION

REGION Network 3: Rotor Overspeed Alarm
   // Activate when rotor speed exceeds the Max setpoint.
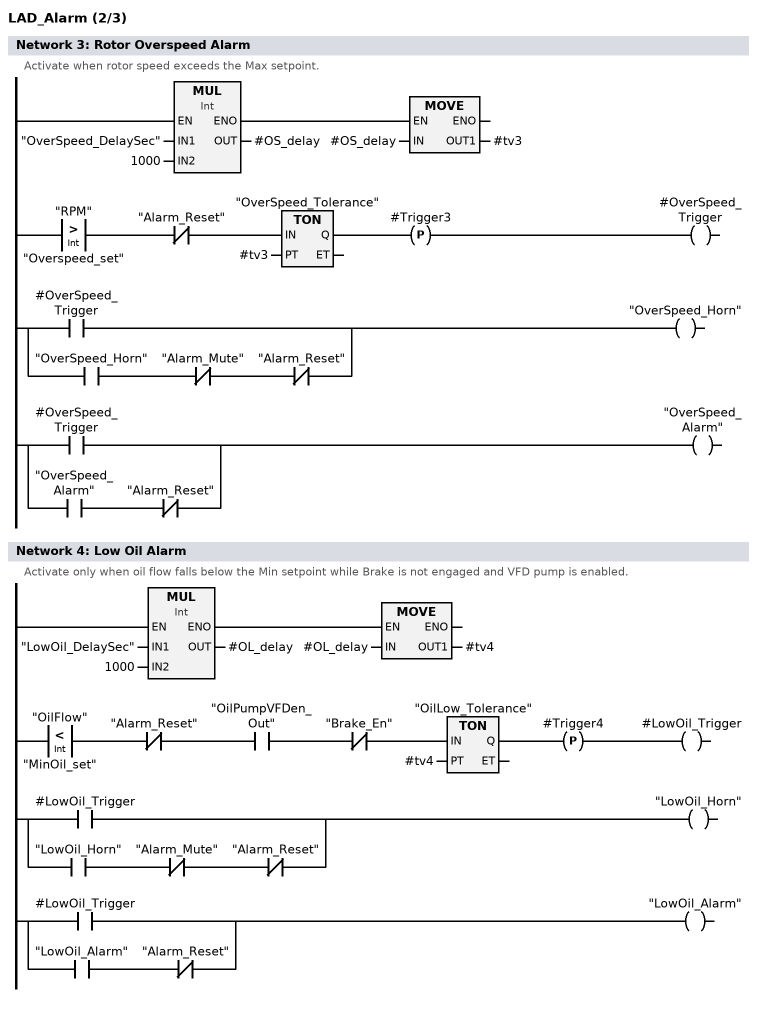
   #OS_delay := "OverSpeed_DelaySec" * 1000;
   #tv3 := #OS_delay;
   "OverSpeed_Tolerance".TON(IN := ("RPM" > "Overspeed_set") AND NOT "Alarm_Reset", PT := #tv3);
   #_w1 := "OverSpeed_Tolerance".Q AND NOT #Trigger3;   // rising edge
   #Trigger3 := "OverSpeed_Tolerance".Q;
   #OverSpeed_Trigger := #_w1;
   "OverSpeed_Horn" := #OverSpeed_Trigger OR ("OverSpeed_Horn" AND NOT "Alarm_Mute" AND NOT "Alarm_Reset");
   "OverSpeed_Alarm" := #OverSpeed_Trigger OR ("OverSpeed_Alarm" AND NOT "Alarm_Reset");
END_REGION

REGION Network 4: Low Oil Alarm
   // Activate only when oil flow falls below the Min setpoint while Brake is not engaged and VFD pump is enabled.
   #OL_delay := "LowOil_DelaySec" * 1000;
   #tv4 := #OL_delay;
   "OilLow_Tolerance".TON(IN := ("OilFlow" < "MinOil_set") AND NOT "Alarm_Reset" AND "OilPumpVFDen_Out" AND NOT "Brake_En",
                          PT := #tv4);
   #_w1 := "OilLow_Tolerance".Q AND NOT #Trigger4;   // rising edge
   #Trigger4 := "OilLow_Tolerance".Q;
   #LowOil_Trigger := #_w1;
   "LowOil_Horn" := #LowOil_Trigger OR ("LowOil_Horn" AND NOT "Alarm_Mute" AND NOT "Alarm_Reset");
   "LowOil_Alarm" := #LowOil_Trigger OR ("LowOil_Alarm" AND NOT "Alarm_Reset");
END_REGION

REGION Network 5: High Oil Alarm
   // Activate when oil flow exceeds the Max setpoint.
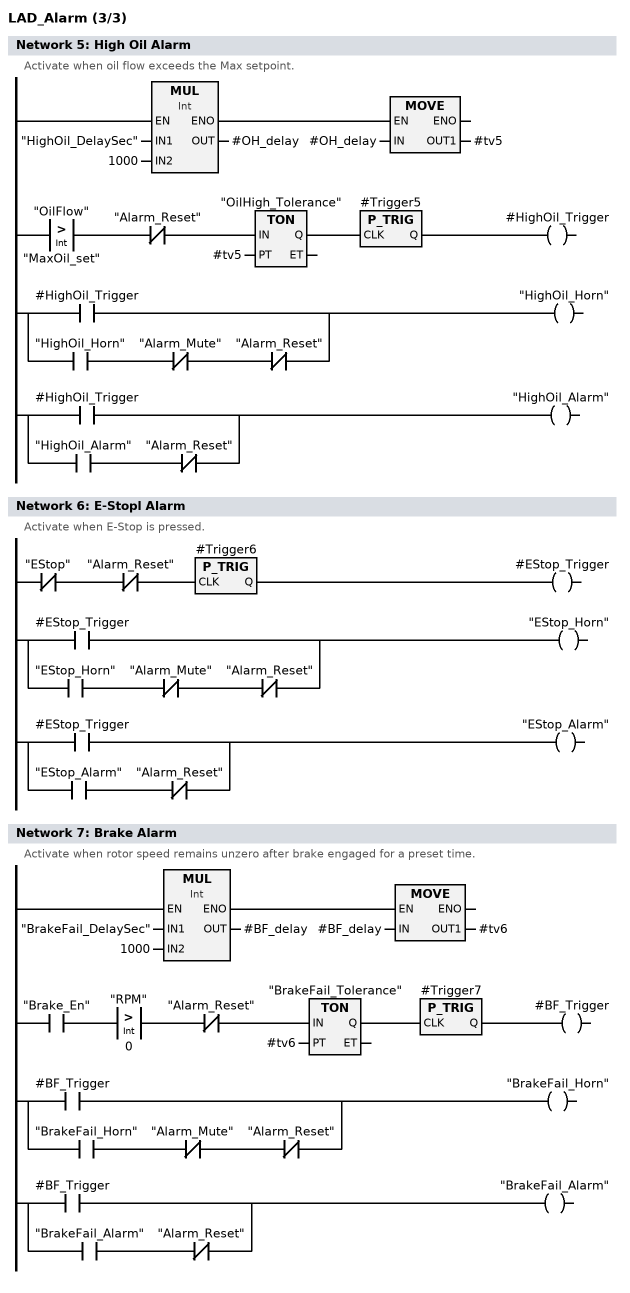
   #OH_delay := "HighOil_DelaySec" * 1000;
   #tv5 := #OH_delay;
   "OilHigh_Tolerance".TON(IN := ("OilFlow" > "MaxOil_set") AND NOT "Alarm_Reset", PT := #tv5);
   #_w1 := "OilHigh_Tolerance".Q AND NOT #Trigger5;   // rising edge
   #Trigger5 := "OilHigh_Tolerance".Q;
   #HighOil_Trigger := #_w1;
   "HighOil_Horn" := #HighOil_Trigger OR ("HighOil_Horn" AND NOT "Alarm_Mute" AND NOT "Alarm_Reset");
   "HighOil_Alarm" := #HighOil_Trigger OR ("HighOil_Alarm" AND NOT "Alarm_Reset");
END_REGION

REGION Network 6: E-Stopl Alarm
   // Activate when E-Stop is pressed.
   RUNG wire#powerrail
      I_Contact( "EStop" )
      I_Contact( "Alarm_Reset" )
      P_Trig( #Trigger6 )
      Coil( #EStop_Trigger )
   END_RUNG
   RUNG wire#powerrail
      Contact( #EStop_Trigger )
      wire#w1
      Coil( "EStop_Horn" )
   END_RUNG
   RUNG wire#powerrail
      Contact( "EStop_Horn" )
      I_Contact( "Alarm_Mute" )
      I_Contact( "Alarm_Reset" )
   END_RUNG wire#w1
   RUNG wire#powerrail
      Contact( #EStop_Trigger )
      wire#w2
      Coil( "EStop_Alarm" )
   END_RUNG
   RUNG wire#powerrail
      Contact( "EStop_Alarm" )
      I_Contact( "Alarm_Reset" )
   END_RUNG wire#w2
   // the same network as SCL:
   #_w1 := NOT "EStop" AND NOT "Alarm_Reset";
   #_w2 := #_w1 AND NOT #Trigger6;   // rising edge
   #Trigger6 := #_w1;
   #EStop_Trigger := #_w2;
   "EStop_Horn" := #EStop_Trigger OR ("EStop_Horn" AND NOT "Alarm_Mute" AND NOT "Alarm_Reset");
   "EStop_Alarm" := #EStop_Trigger OR ("EStop_Alarm" AND NOT "Alarm_Reset");
END_REGION

REGION Network 7: Brake Alarm
   // Activate when rotor speed remains unzero after brake engaged for a preset time.
   #BF_delay := "BrakeFail_DelaySec" * 1000;
   #tv6 := #BF_delay;
   "BrakeFail_Tolerance".TON(IN := "Brake_En" AND ("RPM" > 0) AND NOT "Alarm_Reset", PT := #tv6);
   #_w1 := "BrakeFail_Tolerance".Q AND NOT #Trigger7;   // rising edge
   #Trigger7 := "BrakeFail_Tolerance".Q;
   #BF_Trigger := #_w1;
   "BrakeFail_Horn" := #BF_Trigger OR ("BrakeFail_Horn" AND NOT "Alarm_Mute" AND NOT "Alarm_Reset");
   "BrakeFail_Alarm" := #BF_Trigger OR ("BrakeFail_Alarm" AND NOT "Alarm_Reset");
END_REGION
END_FUNCTION_BLOCK

FUNCTION_BLOCK "FBD_Alarm"   // FB11, FBD
TITLE = Alarms in FBD
{ S7_Optimized_Access := 'TRUE' }
VERSION : 0.1
// When any alarm is triggered, the alert horn will sound. 
// The tolerance time of each alarm can be modified individually. 
// MUL is used to convert sec to ms. MOVE is used to force datatype convert.
// (DInt can be used for longer delays)
   VAR
      Trigger1 : Bool;
      Trigger2 : Bool;
      Trigger3 : Bool;
      Trigger4 : Bool;
      Trigger5 : Bool;
      Trigger6 : Bool;
      Trigger7 : Bool;
   END_VAR
   VAR_TEMP
      OC_delay : Int;
      tv1 : Time;
      OverCurrent_Trigger : Bool;
      HT_delay : Int;
      tv2 : Time;
      OilTempMax_Trigger : Bool;
      OS_delay : Int;
      tv3 : Time;
      OverSpeed_Trigger : Bool;
      OL_delay : Int;
      tv4 : Time;
      LowOil_Trigger : Bool;
      OH_delay : Int;
      tv5 : Time;
      HighOil_Trigger : Bool;
      EStop_Trigger : Bool;
      BF_delay : Int;
      tv6 : Time;
      BF_Trigger : Bool;
   END_VAR
   VAR_TEMP   // added for the SCL form of the ladder/FBD networks
      _w1 : Bool;
      _w2 : Bool;
   END_VAR
BEGIN

REGION Network 1: Overcurrent Alarm
   // Activate when current exceeds the Max setpoint.
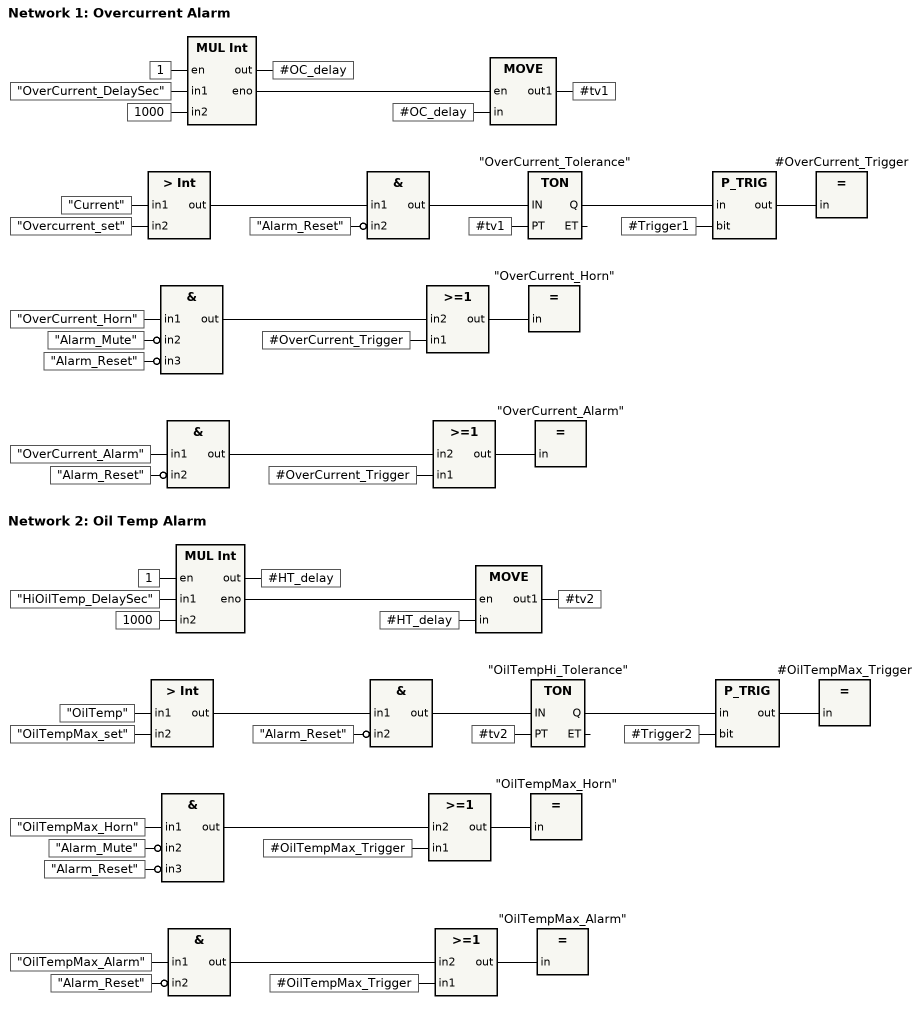
   IF 1 THEN
       #OC_delay := "OverCurrent_DelaySec" * 1000;
       #tv1 := #OC_delay;
   END_IF;
   "OverCurrent_Tolerance".TON(IN := ("Current" > "Overcurrent_set") AND NOT "Alarm_Reset", PT := #tv1);
   #_w1 := "OverCurrent_Tolerance".Q AND NOT #Trigger1;   // rising edge
   #Trigger1 := "OverCurrent_Tolerance".Q;
   #OverCurrent_Trigger := #_w1;
   "OverCurrent_Horn" := ("OverCurrent_Horn" AND NOT "Alarm_Mute" AND NOT "Alarm_Reset") OR #OverCurrent_Trigger;
   "OverCurrent_Alarm" := ("OverCurrent_Alarm" AND NOT "Alarm_Reset") OR #OverCurrent_Trigger;
END_REGION

REGION Network 2: Oil Temp Alarm
   // Activate when oil temperature exceeds the Max setpoint.
   IF 1 THEN
       #HT_delay := "HiOilTemp_DelaySec" * 1000;
       #tv2 := #HT_delay;
   END_IF;
   "OilTempHi_Tolerance".TON(IN := ("OilTemp" > "OilTempMax_set") AND NOT "Alarm_Reset", PT := #tv2);
   #_w1 := "OilTempHi_Tolerance".Q AND NOT #Trigger2;   // rising edge
   #Trigger2 := "OilTempHi_Tolerance".Q;
   #OilTempMax_Trigger := #_w1;
   "OilTempMax_Horn" := ("OilTempMax_Horn" AND NOT "Alarm_Mute" AND NOT "Alarm_Reset") OR #OilTempMax_Trigger;
   "OilTempMax_Alarm" := ("OilTempMax_Alarm" AND NOT "Alarm_Reset") OR #OilTempMax_Trigger;
END_REGION

REGION Network 3: Rotor Overspeed Alarm
   // Activate when rotor speed exceeds the Max setpoint.
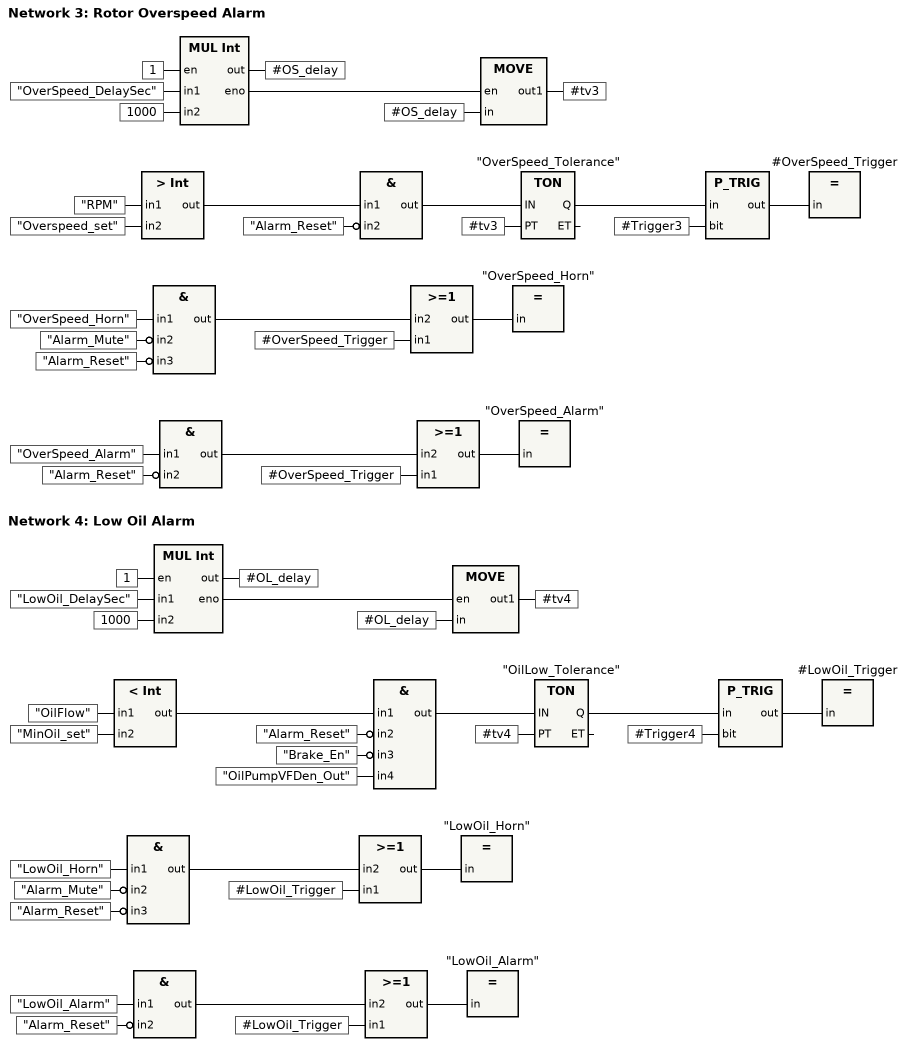
   IF 1 THEN
       #OS_delay := "OverSpeed_DelaySec" * 1000;
       #tv3 := #OS_delay;
   END_IF;
   "OverSpeed_Tolerance".TON(IN := ("RPM" > "Overspeed_set") AND NOT "Alarm_Reset", PT := #tv3);
   #_w1 := "OverSpeed_Tolerance".Q AND NOT #Trigger3;   // rising edge
   #Trigger3 := "OverSpeed_Tolerance".Q;
   #OverSpeed_Trigger := #_w1;
   "OverSpeed_Horn" := ("OverSpeed_Horn" AND NOT "Alarm_Mute" AND NOT "Alarm_Reset") OR #OverSpeed_Trigger;
   "OverSpeed_Alarm" := ("OverSpeed_Alarm" AND NOT "Alarm_Reset") OR #OverSpeed_Trigger;
END_REGION

REGION Network 4: Low Oil Alarm
   // Activate only when oil flow falls below the Min setpoint while Brake is not engaged and VFD pump is enabled.
   IF 1 THEN
       #OL_delay := "LowOil_DelaySec" * 1000;
       #tv4 := #OL_delay;
   END_IF;
   "OilLow_Tolerance".TON(IN := ("OilFlow" < "MinOil_set") AND NOT "Alarm_Reset" AND NOT "Brake_En" AND "OilPumpVFDen_Out",
                          PT := #tv4);
   #_w1 := "OilLow_Tolerance".Q AND NOT #Trigger4;   // rising edge
   #Trigger4 := "OilLow_Tolerance".Q;
   #LowOil_Trigger := #_w1;
   "LowOil_Horn" := ("LowOil_Horn" AND NOT "Alarm_Mute" AND NOT "Alarm_Reset") OR #LowOil_Trigger;
   "LowOil_Alarm" := ("LowOil_Alarm" AND NOT "Alarm_Reset") OR #LowOil_Trigger;
END_REGION

REGION Network 5: High Oil Alarm
   // Activate when oil flow exceeds the Max setpoint.
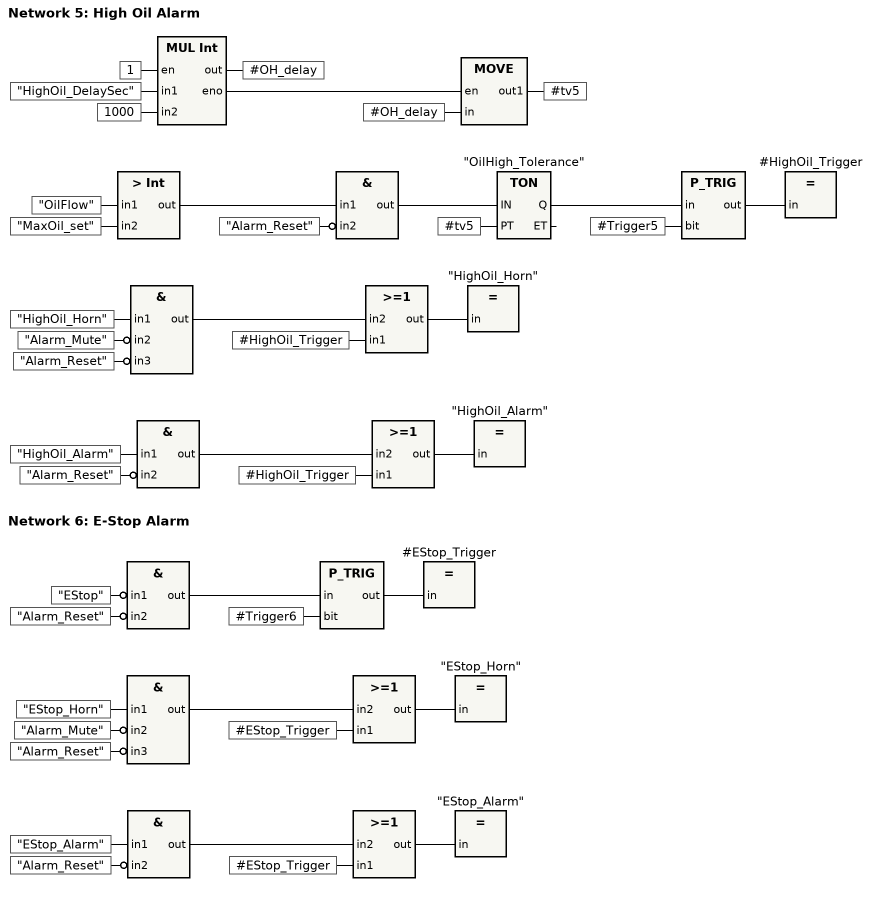
   IF 1 THEN
       #OH_delay := "HighOil_DelaySec" * 1000;
       #tv5 := #OH_delay;
   END_IF;
   "OilHigh_Tolerance".TON(IN := ("OilFlow" > "MaxOil_set") AND NOT "Alarm_Reset", PT := #tv5);
   #_w1 := "OilHigh_Tolerance".Q AND NOT #Trigger5;   // rising edge
   #Trigger5 := "OilHigh_Tolerance".Q;
   #HighOil_Trigger := #_w1;
   "HighOil_Horn" := ("HighOil_Horn" AND NOT "Alarm_Mute" AND NOT "Alarm_Reset") OR #HighOil_Trigger;
   "HighOil_Alarm" := ("HighOil_Alarm" AND NOT "Alarm_Reset") OR #HighOil_Trigger;
END_REGION

REGION Network 6: E-Stop Alarm
   // Activate when E-Stop is pressed.
   #_w1 := NOT "EStop" AND NOT "Alarm_Reset";
   #_w2 := #_w1 AND NOT #Trigger6;   // rising edge
   #Trigger6 := #_w1;
   #EStop_Trigger := #_w2;
   "EStop_Horn" := ("EStop_Horn" AND NOT "Alarm_Mute" AND NOT "Alarm_Reset") OR #EStop_Trigger;
   "EStop_Alarm" := ("EStop_Alarm" AND NOT "Alarm_Reset") OR #EStop_Trigger;
END_REGION

REGION Network 7: Brake Fail Alarm
   // Activate when rotor speed remains unzero after brake engaged for a preset time.
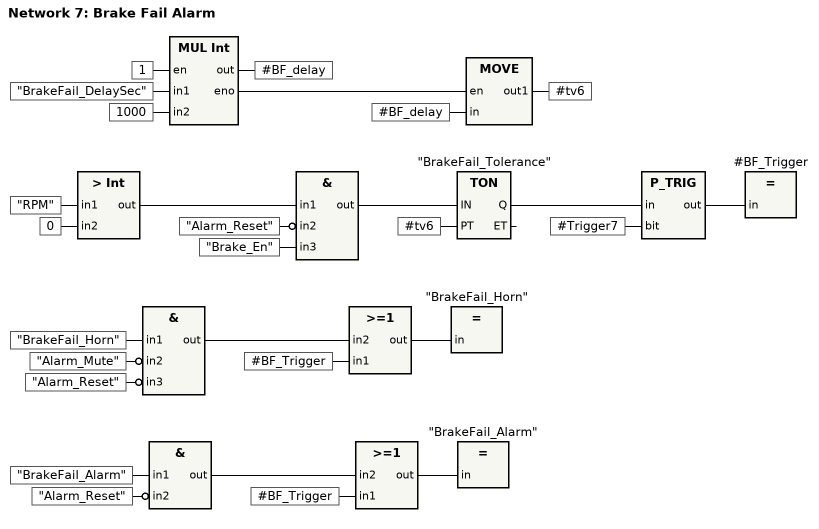
   IF 1 THEN
       #BF_delay := "BrakeFail_DelaySec" * 1000;
       #tv6 := #BF_delay;
   END_IF;
   "BrakeFail_Tolerance".TON(IN := ("RPM" > 0) AND NOT "Alarm_Reset" AND "Brake_En", PT := #tv6);
   #_w1 := "BrakeFail_Tolerance".Q AND NOT #Trigger7;   // rising edge
   #Trigger7 := "BrakeFail_Tolerance".Q;
   #BF_Trigger := #_w1;
   "BrakeFail_Horn" := ("BrakeFail_Horn" AND NOT "Alarm_Mute" AND NOT "Alarm_Reset") OR #BF_Trigger;
   "BrakeFail_Alarm" := ("BrakeFail_Alarm" AND NOT "Alarm_Reset") OR #BF_Trigger;
END_REGION
END_FUNCTION_BLOCK

FUNCTION_BLOCK "SCL_Alarm"   // FB12, SCL
{ S7_Optimized_Access := 'TRUE' }
VERSION : 0.1
   VAR_TEMP
      OC_Delay : Int;
      OverCurrent_Trigger : Bool;
      tv1 : Time;
      OL_Delay : Int;
      tv4 : Time;
      LowOil_Trigger : Bool;
      TimerStart4 : Bool;
      TimerStart1 : Bool;
      HT_Delay : Int;
      tv2 : Time;
      TimerStart2 : Bool;
      OilTempMax_Trigger : Bool;
      OS_Delay : Int;
      OverSpeed_Trigger : Bool;
      tv3 : Time;
      TimerStart3 : Bool;
      OH_Delay : Int;
      tv5 : Time;
      TimerStart5 : Bool;
      HighOil_Trigger : Bool;
      EStop_Trigger : Bool;
      BF_Delay : Int;
      tv6 : Time;
      TimerStart6 : Bool;
      BF_Trigger : Bool;
   END_VAR
BEGIN
   // Alarms in SCL
       // When any alarm is triggered, the alert horn will sound. 
       // The tolerance Time OF each alarm can be modified individually.
       // *1000 is used TO convert sec TO ms. INT_TO_TIME is used TO force datatype convert.
       //(DInt can be used for longer delays.)

   // Overcurrent Alarm
       // Activate when "Current" exceeds the Max setpoint.
       #OC_Delay := "OverCurrent_DelaySec" * 1000;
       #tv1 := INT_TO_TIME(#OC_Delay);

       #TimerStart1 := "Current" > "Overcurrent_set" AND NOT "Alarm_Reset"  AND NOT "OverCurrent_Alarm";
       "OverCurrent_Tolerance".TON(IN := #TimerStart1,
                                   PT := #tv1,
                                   Q => #OverCurrent_Trigger);

       IF #OverCurrent_Trigger THEN
           "OverCurrent_Horn" := 1;
           "OverCurrent_Alarm" := 1;
       END_IF;
       IF "OverCurrent_Alarm" AND "Alarm_Mute" THEN
           "OverCurrent_Horn" := 0;
       END_IF;
       IF "OverCurrent_Alarm" AND "Alarm_Reset" THEN
           "OverCurrent_Alarm" := 0;
           "OverCurrent_Horn" := 0;
       END_IF;


   // Oil Temp Alarm
       // Activate when oil temperature exceeds the Max setpoint.
       #HT_Delay := "HiOilTemp_DelaySec" * 1000;
       #tv2 := INT_TO_TIME(#HT_Delay);

       #TimerStart2 := "OilTemp" > "OilTempMax_set" AND NOT "Alarm_Reset" AND NOT "OilTempMax_Alarm";
       "OilTempHi_Tolerance".TON(IN := #TimerStart2,
                                 PT := #tv2,
                                 Q => #OilTempMax_Trigger);

       IF #OilTempMax_Trigger THEN
           "OilTempMax_Horn" := 1;
           "OilTempMax_Alarm" := 1;
       END_IF;
       IF "OilTempMax_Alarm" AND "Alarm_Mute" THEN
           "OilTempMax_Horn" := 0;
       END_IF;
       IF "OilTempMax_Alarm" AND "Alarm_Reset" THEN
           "OilTempMax_Alarm" := 0;
           "OilTempMax_Horn" := 0;
       END_IF;


   // Rotor Overspeed Alarm
       // Activate when rotor speed exceeds the Max setpoint.
       #OS_Delay := "OverSpeed_DelaySec" * 1000;
       #tv3 := INT_TO_TIME(#OS_Delay);

       #TimerStart3 := "RPM" > "Overspeed_set" AND NOT "Alarm_Reset" AND NOT "OverSpeed_Alarm";
       "OverSpeed_Tolerance".TON(IN := #TimerStart3,
                                 PT := #tv3,
                                 Q => #OverSpeed_Trigger);

       IF #OverSpeed_Trigger THEN
           "OverSpeed_Horn" := 1;
           "OverSpeed_Alarm" := 1;
       END_IF;
       IF "OverSpeed_Alarm" AND "Alarm_Mute" THEN
           "OverSpeed_Horn" := 0;
       END_IF;
       IF "OverSpeed_Alarm" AND "Alarm_Reset" THEN
           "OverSpeed_Alarm" := 0;
           "OverSpeed_Horn" := 0;
       END_IF;


   // Low Oil Alarm
       // Activate only when oil flow falls below the Min setpoint while Brake is not engaged and VFD pump is enabled.
       #OL_Delay := "LowOil_DelaySec" * 1000;
       #tv4 := INT_TO_TIME(#OL_Delay);

       #TimerStart4 := "OilFlow" < "MinOil_set" AND NOT "Alarm_Reset" AND NOT "Brake_En" AND "OilPumpVFDen_Out" AND NOT "LowOil_Alarm";
       "OilLow_Tolerance".TON(IN := #TimerStart4,
                              PT := #tv4,
                              Q => #LowOil_Trigger);

       IF #LowOil_Trigger THEN
           "LowOil_Horn" := 1;
           "LowOil_Alarm" := 1;
       END_IF;
       IF "LowOil_Alarm" AND "Alarm_Mute" THEN
           "LowOil_Horn" := 0;
       END_IF;
       IF "LowOil_Alarm" AND "Alarm_Reset" THEN
           "LowOil_Alarm" := 0;
           "LowOil_Horn" := 0;
       END_IF;


   // High Oil Alarm
       // Activate when oil flow exceeds the Max setpoint.
       #OH_Delay := "HighOil_DelaySec" * 1000;
       #tv5 := INT_TO_TIME(#OH_Delay);

       #TimerStart5 := "OilFlow" > "MaxOil_set" AND NOT "Alarm_Reset" AND NOT "HighOil_Alarm";
       "OilHigh_Tolerance".TON(IN := #TimerStart5,
                                 PT := #tv5,
                                 Q => #HighOil_Trigger);

       IF #HighOil_Trigger THEN
           "HighOil_Horn" := 1;
           "HighOil_Alarm" := 1;
       END_IF;
       IF "HighOil_Alarm" AND "Alarm_Mute" THEN
           "HighOil_Horn" := 0;
       END_IF;
       IF "HighOil_Alarm" AND "Alarm_Reset" THEN
           "HighOil_Alarm" := 0;
           "HighOil_Horn" := 0;
       END_IF;


   // E-Stop Alarm
       // Activate when E-Stop is pressed.
       #EStop_Trigger := NOT "EStop" AND NOT "Alarm_Reset" AND NOT "EStop_Alarm";

       IF #EStop_Trigger THEN
           "EStop_Horn" := 1;
           "EStop_Alarm" := 1;
       END_IF;
       IF "EStop_Alarm" AND "Alarm_Mute" THEN
           "EStop_Horn" := 0;
       END_IF;
       IF "EStop_Alarm" AND "Alarm_Reset" THEN
           "EStop_Alarm" := 0;
           "EStop_Horn" := 0;
       END_IF;


   // Brake Fail Alarm
       // Activate when rotor speed remains unzero after brake engaged for a preset time.
       #BF_Delay := "BrakeFail_DelaySec" * 1000;
       #tv6 := INT_TO_TIME(#BF_Delay);

       #TimerStart6 := "RPM" > 0 AND "Brake_En" AND NOT "Alarm_Reset" AND NOT "BrakeFail_Alarm";
       "BrakeFail_Tolerance".TON(IN := #TimerStart6,
                             PT := #tv6,
                             Q => #BF_Trigger);

       IF #BF_Trigger THEN
           "BrakeFail_Horn" := 1;
           "BrakeFail_Alarm" := 1;
       END_IF;
       IF "BrakeFail_Alarm" AND "Alarm_Mute" THEN
           "BrakeFail_Horn" := 0;
       END_IF;
       IF "BrakeFail_Alarm" AND "Alarm_Reset" THEN
           "BrakeFail_Alarm" := 0;
           "BrakeFail_Horn" := 0;
       END_IF;
END_FUNCTION_BLOCK

FUNCTION_BLOCK "STL_Alarm"   // FB13, STL
TITLE = Alarms in STL
{ S7_Optimized_Access := 'TRUE' }
VERSION : 0.1
// When any alarm is triggered, the alert horn will sound. 
// The tolerance time of each alarm can be modified individually. 
// *D is used to convert sec to ms. ITD is used to force datatype convert.
// DInt type is directly used here for the TON timer.
   VAR
      os1 : Bool;
      os2 : Bool;
      os3 : Bool;
      os4 : Bool;
      os5 : Bool;
      os6 : Bool;
      os7 : Bool;
      os8 : Bool;
      os9 : Bool;
      os10 : Bool;
      os11 : Bool;
      os12 : Bool;
      os13 : Bool;
      os14 : Bool;
      os15 : Bool;
      Overcurrent_Muted : Bool;
   END_VAR
   VAR_TEMP
      tv1 : Time;
      tv2 : Time;
      tv3 : Time;
      tv4 : Time;
      tv5 : Time;
      tv6 : Time;
      OverCurrent_Trigger : Bool;
      OilTempMax_Trigger : Bool;
      OverSpeed_Trigger : Bool;
      LowOil_Trigger : Bool;
      HighOil_Trigger : Bool;
      EStop_Trigger : Bool;
      BF_Trigger : Bool;
   END_VAR
BEGIN

REGION Network 1: Overcurrent Alarm
   // Activate when current exceeds the Max setpoint.
         A     "Alarm_Reset";
         FP    #os1;
         JC    ResetAlarmOC;
         CLR;
         A     "Alarm_Mute";
         FP    #os2;
         JC    MuteAlarmOC;
         CLR;

         L     "Current";
         L     "Overcurrent_set";
         >I;
         JC    TimerOC;
         JU    OilTemp;

   TimerOC:L     "OverCurrent_DelaySec";
         ITD;
         L     DINT#1000;
         *D;
         T     #tv1;
         CALL  TON, "OverCurrent_Tolerance"
         ( IN := 1,
           PT := #tv1,
           Q  := #OverCurrent_Trigger,
           ET :=
         );
         A     #OverCurrent_Trigger;
         AN    "OverCurrent_Alarm";
         JC    SetAlarmOC;
         JU    OilTemp;

   SetAlarmOC:SET;
         S     "OverCurrent_Alarm";
         S     "OverCurrent_Horn";
         JU    OilTemp;

   ResetAlarmOC:R     "OverCurrent_Alarm";
         R     "OverCurrent_Horn";
         CALL  RESET_TIMER
         ( "TIMER" := "OverCurrent_Tolerance"
         );
         JU    OilTemp;

   MuteAlarmOC:R     "OverCurrent_Horn";
END_REGION

REGION Network 2: Oil Temp Alarm
   // Activate when oil temperature exceeds the Max setpoint.
   OilTemp:A     "Alarm_Reset";
         FP    #os3;
         JC    ResetAlarmHT;
         CLR;
         A     "Alarm_Mute";
         FP    #os4;
         JC    MuteAlarmHT;
         CLR;

         L     "OilTemp";
         L     "OilTempMax_set";
         >I;
         JC    TimerHT;
         JU    Rotor;

   TimerHT:L     "HiOilTemp_DelaySec";
         ITD;
         L     DINT#1000;
         *D;
         T     #tv2;
         CALL  TON , "OilTempHi_Tolerance"
         ( IN := 1,
           PT := #tv2,
           Q  := #OilTempMax_Trigger,
           ET :=
         );
         A     #OilTempMax_Trigger;
         AN    "OilTempMax_Alarm";
         JC    SetAlarmHT;
         JU    Rotor;

   SetAlarmHT:SET;
         S     "OilTempMax_Alarm";
         S     "OilTempMax_Horn";
         JU    Rotor;

   ResetAlarmHT:R     "OilTempMax_Alarm";
         R     "OilTempMax_Horn";
         CALL  RESET_TIMER
         ( "TIMER" := "OilTempHi_Tolerance"
         );
         JU    Rotor;

   MuteAlarmHT:R     "OilTempMax_Horn";
END_REGION

REGION Network 3: Rotor Overspeed Alarm
   // Activate when rotor speed exceeds the Max setpoint.
   Rotor:A     "Alarm_Reset";
         FP    #os5;
         JC    ResetAlarmOS;
         CLR;
         A     "Alarm_Mute";
         FP    #os6;
         JC    MuteAlarmOS;
         CLR;

         L     "RPM";
         L     "Overspeed_set";
         >I;
         AN    "Alarm_Reset";
         JC    TimerOS;
         JU    LowOil;

   TimerOS:L     "OverSpeed_DelaySec";
         ITD;
         L     DINT#1000;
         *D;
         T     #tv3;
         CALL  TON , "OverSpeed_Tolerance"
         ( IN := 1,
           PT := #tv3,
           Q  := #OverSpeed_Trigger,
           ET :=
         );
         A     #OverSpeed_Trigger;
         AN    "OverSpeed_Alarm";
         JC    SetAlarmOS;
         JU    LowOil;

   SetAlarmOS:SET;
         S     "OverSpeed_Alarm";
         S     "OverSpeed_Horn";
         JU    LowOil;

   ResetAlarmOS:R     "OverSpeed_Alarm";
         R     "OverSpeed_Horn";
         CALL  RESET_TIMER
         ( "TIMER" := "OverSpeed_Tolerance"
         );
         JU    LowOil;

   MuteAlarmOS:R     "OverSpeed_Horn";
END_REGION

REGION Network 4: Low Oil Alarm
   // Activate only when oil flow falls below the Min setpoint while Brake is not engaged and VFD pump is enabled.
   LowOil:A     "Alarm_Reset";
         FP    #os7;
         JC    ResetAlarmOL;
         CLR;
         A     "Alarm_Mute";
         FP    #os8;
         JC    MuteAlarmOL;
         CLR;

         L     "OilFlow";
         L     "MinOil_set";
         <I;
         A     "OilPumpVFDen_Out";
         AN    "Brake_En";
         JC    TimerOL;
         JU    HighOil;

   TimerOL:L     "LowOil_DelaySec";
         ITD;
         L     DINT#1000;
         *D;
         T     #tv4;
         CALL  TON , "OilLow_Tolerance"
         ( IN := 1,
           PT := #tv4,
           Q  := #LowOil_Trigger,
           ET :=
         );
         A     #LowOil_Trigger;
         AN    "LowOil_Alarm";
         JC    SetAlarmOL;
         JU    HighOil;

   SetAlarmOL:SET;
         S     "LowOil_Alarm";
         S     "LowOil_Horn";
         JU    HighOil;

   ResetAlarmOL:R     "LowOil_Alarm";
         R     "LowOil_Horn";
         CALL  RESET_TIMER
         ( "TIMER" := "OilLow_Tolerance"
         );
         JU    HighOil;

   MuteAlarmOL:R     "LowOil_Horn";
END_REGION

REGION Network 5: High Oil Alarm
   // Activate when oil flow exceeds the Max setpoint.
   HighOil:A     "Alarm_Reset";
         FP    #os9;
         JC    ResetAlarmOH;
         CLR;
         A     "Alarm_Mute";
         FP    #os10;
         JC    MuteAlarmOH;
         CLR;

         L     "OilFlow";
         L     "MaxOil_set";
         >I;
         JC    TimerOH;
         JU    Estop;

   TimerOH:L     "HighOil_DelaySec";
         ITD;
         L     DINT#1000;
         *D;
         T     #tv5;
         CALL  TON , "OilHigh_Tolerance"
         ( IN := 1,
           PT := #tv5,
           Q  := #HighOil_Trigger,
           ET :=
         );
         A     #HighOil_Trigger;
         AN    "HighOil_Alarm";
         JC    SetAlarmOH;
         JU    Estop;

   SetAlarmOH:SET;
         S     "HighOil_Alarm";
         S     "HighOil_Horn";
         JU    Estop;

   ResetAlarmOH:R     "HighOil_Alarm";
         R     "HighOil_Horn";
         CALL  RESET_TIMER
         ( "TIMER" := "OilHigh_Tolerance"
         );
         JU    Estop;

   MuteAlarmOH:R     "HighOil_Horn";
END_REGION

REGION Network 6: E-Stop Alarm
   // Activate when E-Stop is pressed.
   Estop:A     "Alarm_Reset";
         FP    #os11;
         JC    ResetAlarmES;
         CLR;
         A     "Alarm_Mute";
         FP    #os12;
         JC    MuteAlarmES;
         CLR;

         AN    "EStop";
         AN    "Alarm_Reset";
         AN    "EStop_Alarm";
         JC    SetAlarmES;
         JU    Brake;


   SetAlarmES:SET;
         S     "EStop_Alarm";
         S     "EStop_Horn";
         JU    Brake;

   ResetAlarmES:R     "EStop_Alarm";
         R     "EStop_Horn";
         JU    Brake;

   MuteAlarmES:R     "EStop_Horn";
END_REGION

REGION Network 7
   Brake:A     "Alarm_Reset";
         FP    #os13;
         JC    ResetAlarmBF;
         CLR;
         A     "Alarm_Mute";
         FP    #os14;
         JC    MuteAlarmBF;
         CLR;

         L     "RPM";
         L     0;
         >I;
         A     "Brake_En";
         AN    "Alarm_Reset";
         JC    TimerBF;
         JU    End;

   TimerBF:L     "BrakeFail_DelaySec";
         ITD;
         L     DINT#1000;
         *D;
         T     #tv6;
         CALL  TON , "BrakeFail_Tolerance"
         ( IN := 1,
           PT := #tv6,
           Q  := #BF_Trigger,
           ET :=
         );
         A     #BF_Trigger;
         AN    "BrakeFail_Alarm";
         JC    SetAlarmBF;
         JU    End;

   SetAlarmBF:SET;
         S     "BrakeFail_Alarm";
         S     "BrakeFail_Horn";
         JU    End;

   ResetAlarmBF:R     "BrakeFail_Alarm";
         R     "BrakeFail_Horn";
         CALL  RESET_TIMER
         ( "TIMER" := "BrakeFail_Tolerance"
         );
         JU    End;

   MuteAlarmBF:R     "BrakeFail_Horn";

   End:  BE;
END_REGION
END_FUNCTION_BLOCK

FUNCTION_BLOCK "LAD_Modes"   // FB14, LAD
TITLE = System Modes in Ladder Diagram
{ S7_Optimized_Access := 'TRUE' }
VERSION : 0.1
// Warmup – When Start pushbutton is pressed, the sequence begins with this step. Allow the rotor to turn at a speed somethere between 20 and 50 RPMs and run the oil pump at some low output level (2-10 GPM) until the oil temp reaches 150 degrees. Once we’ve maintained at least 150 degrees
// for 10 seconds, we want to transition into the next mode.
// 
// Stabilize – Generator should speed up until desired kW output is attained. Once we’re stable within 5kW (+/-) of the setpoint for at least 10 seconds, we should transition into the next mode.
// 
// Generation – Keep everything running and close the interlock.
// 
// Cooldown – Once the Stop button has been pushed, open the interlock, slow the rotor to between 20 and 50 RPMs and maintain a high oil flow until the oil temp is below 150 degrees. Once we’re below for 10 seconds, we transition into Idle mode.
// 
// Idle – Interlock and baffle are deenergized and brake is engaged.
// 
// Fault – When we hit an alarm, the sequence should be aborted according to the alarm details (in the Alarms section), and we should go into Fault mode (which is not part of our sequence).
   VAR
      trigger1 : Bool;
      trigger2 : Bool;
      trigger3 : Bool;
      trigger4 : Bool;
      trigger5 : Bool;
   END_VAR
   VAR_TEMP
      tv1 : Int;
      timer1 : Time;
      tv2 : Int;
      tv3 : Int;
      tv4 : Int;
      timer2 : Time;
      tv5 : Int;
      timer3 : Time;
   END_VAR
   VAR_TEMP   // added for the SCL form of the ladder/FBD networks
      _w1 : Bool;
      _w2 : Bool;
      _w3 : Bool;
   END_VAR
BEGIN

REGION Network 1: Warmup Mode
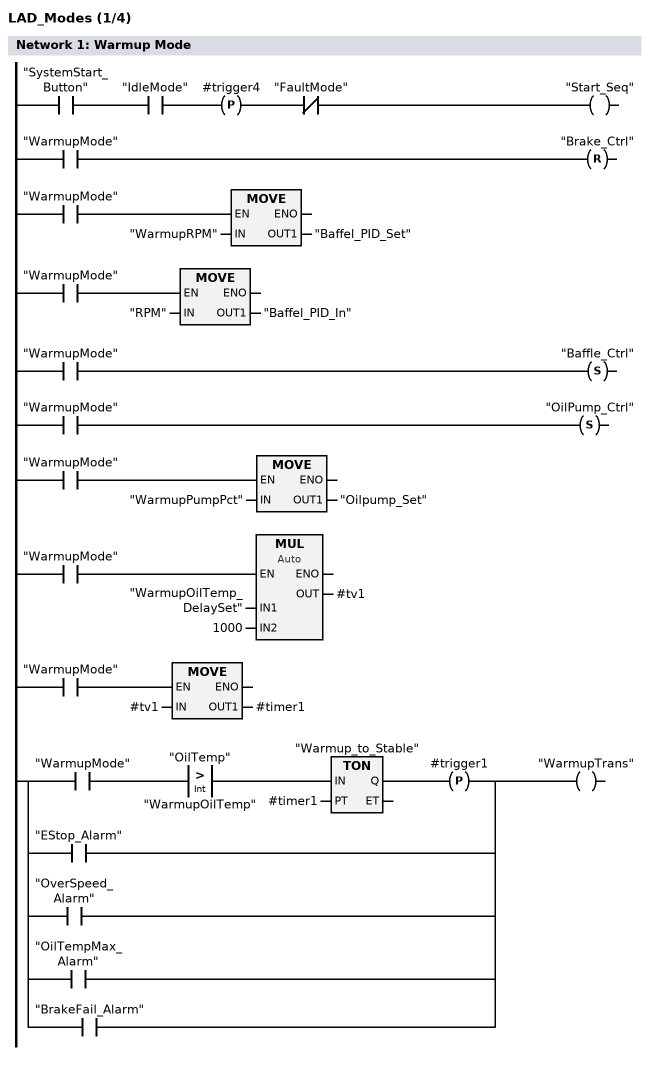
   #_w1 := "SystemStart_Button" AND "IdleMode";
   #_w2 := #_w1 AND NOT #trigger4;   // rising edge
   #trigger4 := #_w1;
   "Start_Seq" := #_w2 AND NOT "FaultMode";
   IF "WarmupMode" THEN
       "Brake_Ctrl" := FALSE;
       "Baffel_PID_Set" := "WarmupRPM";
       "Baffel_PID_In" := "RPM";
       "Baffle_Ctrl" := TRUE;
       "OilPump_Ctrl" := TRUE;
       "Oilpump_Set" := "WarmupPumpPct";
       #tv1 := "WarmupOilTemp_DelaySet" * 1000;
       #timer1 := #tv1;
   END_IF;
   "Warmup_to_Stable".TON(IN := "WarmupMode" AND ("OilTemp" > "WarmupOilTemp"), PT := #timer1);
   #_w3 := "Warmup_to_Stable".Q AND NOT #trigger1;   // rising edge
   #trigger1 := "Warmup_to_Stable".Q;
   "WarmupTrans" := #_w3 OR "EStop_Alarm" OR "OverSpeed_Alarm" OR "OilTempMax_Alarm" OR "BrakeFail_Alarm";
END_REGION

REGION Network 2: Stabilize Mode
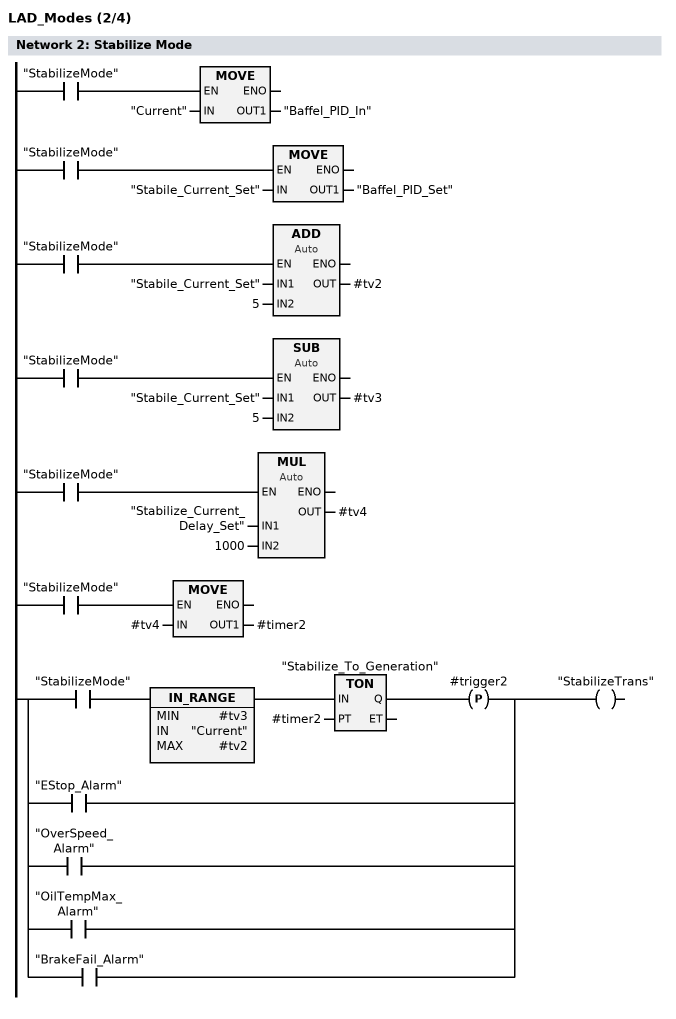
   IF "StabilizeMode" THEN
       "Baffel_PID_In" := "Current";
       "Baffel_PID_Set" := "Stabile_Current_Set";
       #tv2 := "Stabile_Current_Set" + 5;
       #tv3 := "Stabile_Current_Set" - 5;
       #tv4 := "Stabilize_Current_Delay_Set" * 1000;
       #timer2 := #tv4;
   END_IF;
   "Stabilize_To_Generation".TON(IN := "StabilizeMode" AND (#tv3 <= "Current") AND ("Current" <= #tv2),
                           PT := #timer2);
   #_w1 := "Stabilize_To_Generation".Q AND NOT #trigger2;   // rising edge
   #trigger2 := "Stabilize_To_Generation".Q;
   "StabilizeTrans" := #_w1 OR "EStop_Alarm" OR "OverSpeed_Alarm" OR "OilTempMax_Alarm" OR "BrakeFail_Alarm";
END_REGION

REGION Network 3: Generation Mode
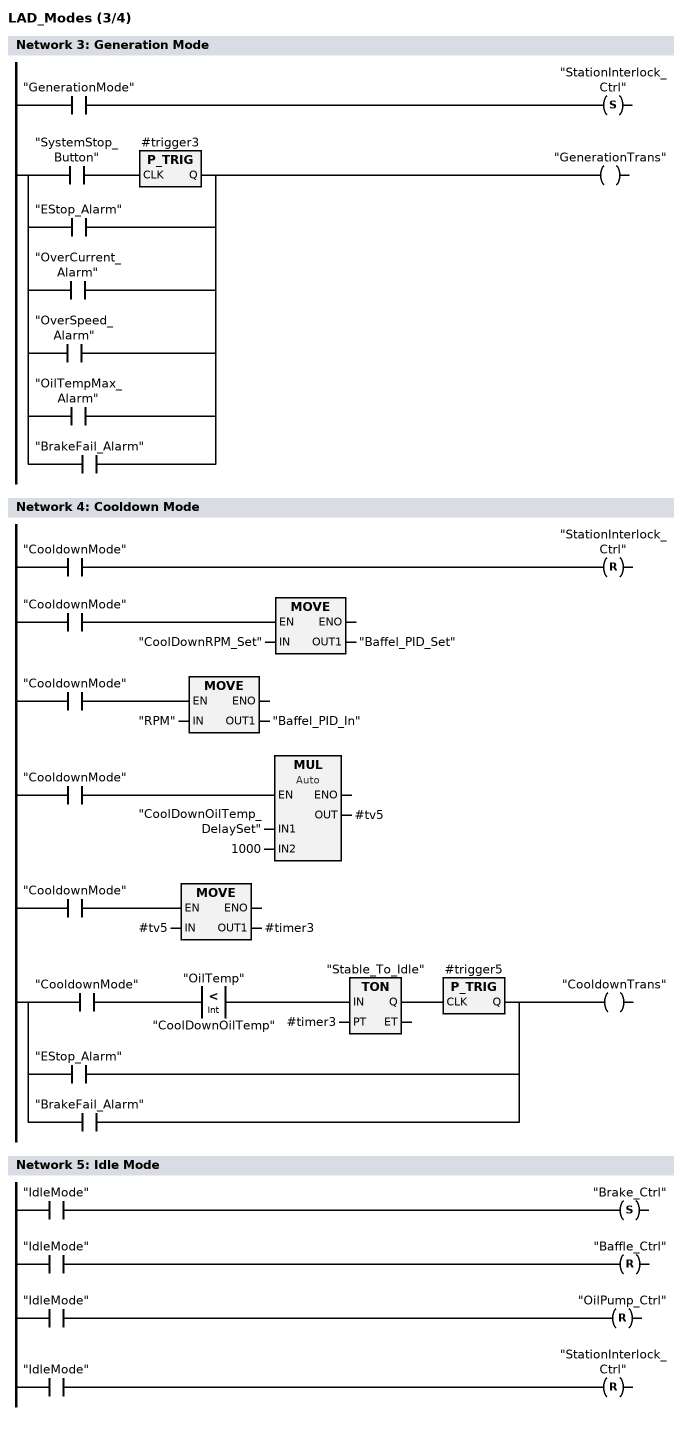
   RUNG wire#powerrail
      Contact( "GenerationMode" )
      S_Coil( "StationInterlock_Ctrl" )
   END_RUNG
   RUNG wire#powerrail
      Contact( "SystemStop_Button" )
      P_Trig( #trigger3 )
      wire#w1
      Coil( "GenerationTrans" )
   END_RUNG
   RUNG wire#powerrail
      Contact( "EStop_Alarm" )
   END_RUNG wire#w1
   RUNG wire#powerrail
      Contact( "OverCurrent_Alarm" )
   END_RUNG wire#w1
   RUNG wire#powerrail
      Contact( "OverSpeed_Alarm" )
   END_RUNG wire#w1
   RUNG wire#powerrail
      Contact( "OilTempMax_Alarm" )
   END_RUNG wire#w1
   RUNG wire#powerrail
      Contact( "BrakeFail_Alarm" )
   END_RUNG wire#w1
   // the same network as SCL:
   IF "GenerationMode" THEN "StationInterlock_Ctrl" := TRUE; END_IF;
   #_w1 := "SystemStop_Button" AND NOT #trigger3;   // rising edge
   #trigger3 := "SystemStop_Button";
   "GenerationTrans" := #_w1 OR "EStop_Alarm" OR "OverCurrent_Alarm" OR "OverSpeed_Alarm" OR "OilTempMax_Alarm" OR "BrakeFail_Alarm";
END_REGION

REGION Network 4: Cooldown Mode
   IF "CooldownMode" THEN
       "StationInterlock_Ctrl" := FALSE;
       "Baffel_PID_Set" := "CoolDownRPM_Set";
       "Baffel_PID_In" := "RPM";
       #tv5 := "CoolDownOilTemp_DelaySet" * 1000;
       #timer3 := #tv5;
   END_IF;
   "Stable_To_Idle".TON(IN := "CooldownMode" AND ("OilTemp" < "CoolDownOilTemp"), PT := #timer3);
   #_w1 := "Stable_To_Idle".Q AND NOT #trigger5;   // rising edge
   #trigger5 := "Stable_To_Idle".Q;
   "CooldownTrans" := #_w1 OR "EStop_Alarm" OR "BrakeFail_Alarm";
END_REGION

REGION Network 5: Idle Mode
   RUNG wire#powerrail
      Contact( "IdleMode" )
      S_Coil( "Brake_Ctrl" )
   END_RUNG
   RUNG wire#powerrail
      Contact( "IdleMode" )
      R_Coil( "Baffle_Ctrl" )
   END_RUNG
   RUNG wire#powerrail
      Contact( "IdleMode" )
      R_Coil( "OilPump_Ctrl" )
   END_RUNG
   RUNG wire#powerrail
      Contact( "IdleMode" )
      R_Coil( "StationInterlock_Ctrl" )
   END_RUNG
   // the same network as SCL:
   IF "IdleMode" THEN
       "Brake_Ctrl" := TRUE;
       "Baffle_Ctrl" := FALSE;
       "OilPump_Ctrl" := FALSE;
       "StationInterlock_Ctrl" := FALSE;
   END_IF;
END_REGION

REGION Network 6: Fault Mode
   // NOT in the sequence
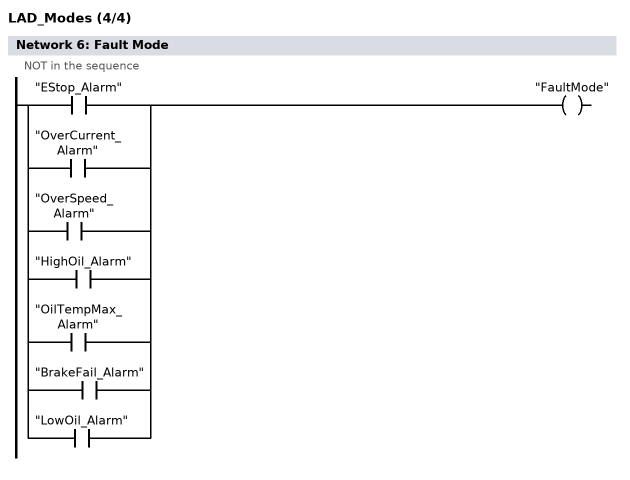
   RUNG wire#powerrail
      Contact( "EStop_Alarm" )
      wire#w1
      Coil( "FaultMode" )
   END_RUNG
   RUNG wire#powerrail
      Contact( "OverCurrent_Alarm" )
   END_RUNG wire#w1
   RUNG wire#powerrail
      Contact( "OverSpeed_Alarm" )
   END_RUNG wire#w1
   RUNG wire#powerrail
      Contact( "HighOil_Alarm" )
   END_RUNG wire#w1
   RUNG wire#powerrail
      Contact( "OilTempMax_Alarm" )
   END_RUNG wire#w1
   RUNG wire#powerrail
      Contact( "BrakeFail_Alarm" )
   END_RUNG wire#w1
   RUNG wire#powerrail
      Contact( "LowOil_Alarm" )
   END_RUNG wire#w1
   // the same network as SCL:
   "FaultMode" := "EStop_Alarm" OR "OverCurrent_Alarm" OR "OverSpeed_Alarm" OR "HighOil_Alarm" OR "OilTempMax_Alarm" OR "BrakeFail_Alarm" OR "LowOil_Alarm";
END_REGION
END_FUNCTION_BLOCK

FUNCTION_BLOCK "SEQ"   // FB15, GRAPH_PLUS
{ S7_Optimized_Access := 'TRUE' }
VERSION : 0.1
   VAR_INPUT
      OFF_SQ : Bool := false;   // Turn sequence off
      INIT_SQ : Bool := false;   // Set sequence to initial state
      ACK_EF : Bool := false;   // Acknowledge all errors and faults
      S_PREV : Bool := false;   // Output previous step in parameter S_NO
      S_NEXT : Bool := false;   // Indicate next step in parameter S_NO
      SW_AUTO : Bool := false;   // Automatic mode
      SW_TAP : Bool := false;   // Semiautomatic/switch with transition
      SW_TOP : Bool := false;   // Semiautomatic/ignore transition
      SW_MAN : Bool := false;   // Manual mode
      S_SEL : Int := 0;   // Select step to be output to S_NO
      S_ON : Bool := false;   // Activate step indicated in S_NO
      S_OFF : Bool := false;   // Disable step indicated in S_NO
      T_PUSH : Bool := false;   // Enable transition to switch in semi automatic mode
   END_VAR
   VAR_OUTPUT
      S_NO : Int := 0;   // Step number
      S_MORE : Bool := false;   // More steps are available and can be shown in S_NO
      S_ACTIVE : Bool := false;   // Step indicated in S_NO is active
      ERR_FLT : Bool := false;   // Interlock or supervision group error
      AUTO_ON : Bool := false;   // Automatic mode is active
      TAP_ON : Bool := false;   // Semiautomatic mode/step with transition enabled
      TOP_ON : Bool := false;   // Semiautomatic mode/ignore transition enabled
      MAN_ON : Bool := false;   // Manual mode is active
   END_VAR
   VAR
      HMI_INFO : Array[0..8] of UInt;
      IF_PAR : G7_IfParPlus_V2;
      RT_DATA : G7_RTDataPlus_V2;   // Internal data area
      Trans1 : G7_TransitionPlus_V2;   // Transition structure
      Trans2 : G7_TransitionPlus_V2;   // Transition structure
      Trans3 : G7_TransitionPlus_V2;   // Transition structure
      Trans4 : G7_TransitionPlus_V2;   // Transition structure
      Trans5 : G7_TransitionPlus_V2;   // Transition structure
      Idle : G7_StepPlus_V2;   // Step structure
      Warmup : G7_StepPlus_V2;   // Step structure
      Stabilize : G7_StepPlus_V2;   // Step structure
      Generation : G7_StepPlus_V2;   // Step structure
      Cooldown : G7_StepPlus_V2;   // Step structure
      SINI : Array[0..1] of USInt;
      LSTT : Array[0..4] of USInt;
      ATAJ : Array[0..4] of USInt;
      ATAB : Array[0..4] of USInt;
      PSTT : Array[0..4] of USInt;
      NSTT : Array[0..4] of USInt;
      ASSJ : Array[0..4] of USInt;
      ASSB : Array[0..4] of USInt;
      PTTS : Array[0..4] of USInt;
      NTTS : Array[0..4] of USInt;
      SW_SQTS : Array[0..4] of USInt;
      SWITCH : Array[0..0] of USInt;
      TVX : Array[0..1] of USInt;
      TTX : Array[0..1] of USInt;
      TSX : Array[0..1] of USInt;
      S00X : Array[0..1] of USInt;
      SOFFX : Array[0..1] of USInt;
      SONX : Array[0..1] of USInt;
      SAX : Array[0..1] of USInt;
      SERRX : Array[0..5] of USInt;
      SMX : Array[0..5] of USInt;
      S0X : Array[0..5] of USInt;
      S1X : Array[0..5] of USInt;
      IL_ALARM_INST : Program_Alarm;
      SUP_ALARM_INST : Program_Alarm;
      STEP_TIME_ALARM_INST : Program_Alarm;
      IEC_TIMER_INST : IEC_TIMER;
      TRANSACTION_FLAG : Bool := false;
   END_VAR
   // SINI[0] := 2;
   // LSTT[0] := 255;
   // LSTT[1] := 255;
   // LSTT[2] := 255;
   // LSTT[3] := 255;
   // ATAJ[1] := 1;
   // ATAJ[2] := 2;
   // ATAJ[3] := 3;
   // ATAJ[4] := 4;
   // ATAB[1] := 1;
   // ATAB[2] := 2;
   // ATAB[3] := 3;
   // ATAB[4] := 4;
   // PSTT[1] := 1;
   // PSTT[2] := 2;
   // PSTT[3] := 3;
   // PSTT[4] := 4;
   // NSTT[0] := 1;
   // NSTT[1] := 2;
   // NSTT[2] := 3;
   // NSTT[3] := 4;
   // ASSJ[1] := 1;
   // ASSJ[2] := 2;
   // ASSJ[3] := 3;
   // ASSJ[4] := 4;
   // ASSB[1] := 1;
   // ASSB[2] := 2;
   // ASSB[3] := 3;
   // ASSB[4] := 4;
   // PTTS[0] := 255;
   // PTTS[2] := 1;
   // PTTS[3] := 2;
   // PTTS[4] := 3;
   // NTTS[1] := 1;
   // NTTS[2] := 2;
   // NTTS[3] := 3;
   // NTTS[4] := 4;
   // TVX[0] := 16#1;
   // TTX[0] := 16#1;
   // TSX[0] := 16#1;
   // S00X[0] := 16#1;
   // SOFFX[0] := 16#1;
   // SONX[0] := 16#1;
   // SAX[0] := 16#1;
   // SERRX[0] := 16#1;
   // SMX[0] := 16#1;
   // S0X[0] := 16#1;
   // S1X[0] := 16#1;
BEGIN
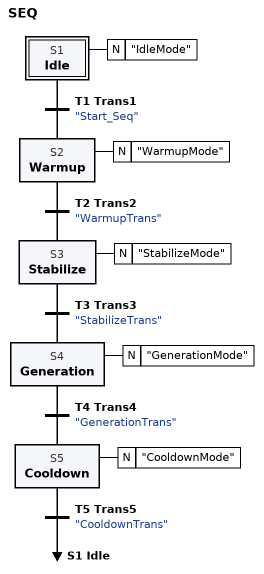
   // sequencer 1
   INITIAL_STEP Idle:   // S1, max time T#10S, warning time T#7S
              N    "IdleMode"
   END_STEP
   TRANSITION Trans1 FROM Idle TO Warmup   // T1
      := "Start_Seq";
   END_TRANSITION
   STEP Warmup:   // S2, max time T#10S, warning time T#7S
              N    "WarmupMode"
   END_STEP
   TRANSITION Trans2 FROM Warmup TO Stabilize   // T2
      := "WarmupTrans";
   END_TRANSITION
   STEP Stabilize:   // S3, max time T#10S, warning time T#7S
              N    "StabilizeMode"
   END_STEP
   TRANSITION Trans3 FROM Stabilize TO Generation   // T3
      := "StabilizeTrans";
   END_TRANSITION
   STEP Generation:   // S4, max time T#10S, warning time T#7S
              N    "GenerationMode"
   END_STEP
   TRANSITION Trans4 FROM Generation TO Cooldown   // T4
      := "GenerationTrans";
   END_TRANSITION
   STEP Cooldown:   // S5, max time T#10S, warning time T#7S
              N    "CooldownMode"
   END_STEP
   TRANSITION Trans5 FROM Cooldown TO Idle   // T5, jump
      := "CooldownTrans";
   END_TRANSITION
END_FUNCTION_BLOCK

FUNCTION "Conversion_func" : Void   // FC1, LAD
{ S7_Optimized_Access := 'TRUE' }
VERSION : 0.1
   VAR_INPUT
      Input_min : Int;
      Input_max : Int;
      Input_value : Int;
      Output_min : Int;
      Output_max : Int;
   END_VAR
   VAR_OUTPUT
      Output_value : Int;
   END_VAR
   VAR_TEMP
      Norm_value : Real;
   END_VAR
BEGIN

REGION Network 1: General Conversion Process
   // Formal: "Normalize + Scale"
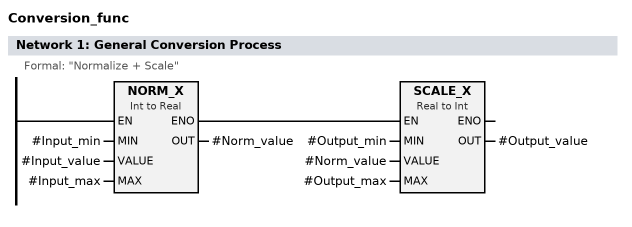
   RUNG wire#powerrail
      { S7_Templates := "[SrcType := Int, DestType := Real]" } Normalize(min := #Input_min, value := #Input_value, max := #Input_max, out => #Norm_value)
      { S7_Templates := "[SrcType := Real, DestType := Int]" } Scale(min := #Output_min, value := #Norm_value, max := #Output_max, out => #Output_value)
   END_RUNG
   // the same network as SCL:
   #Norm_value := NORM_X(MIN := #Input_min, VALUE := #Input_value, MAX := #Input_max);
   #Output_value := SCALE_X(MIN := #Output_min, VALUE := #Norm_value, MAX := #Output_max);
END_REGION
END_FUNCTION

FUNCTION "Conversion_func_rev" : Void   // FC2, LAD
{ S7_Optimized_Access := 'TRUE' }
VERSION : 0.1
   VAR_INPUT
      Input_min : Int;
      Input_max : Int;
      Input_value : Int;
      Output_min : Int;
      Output_max : Int;
   END_VAR
   VAR_OUTPUT
      Output_value : Int;
   END_VAR
   VAR_TEMP
      Norm_value : Real;
      Norm_value_rev : Real;
   END_VAR
BEGIN

REGION Network 1
